C01814=1078.084,-56.704,-56.750,173.466,20.388,153.550
C01815=1078.090,-56.454,-56.762,173.467,20.389,153.550
C01816=1078.097,-56.206,-56.774,173.468,20.391,153.551
C01817=1078.102,-55.955,-56.785,173.470,20.393,153.551
C01818=1078.108,-55.706,-56.797,173.472,20.395,153.551
C01819=1078.115,-55.456,-56.808,173.473,20.397,153.551
C01820=1078.120,-55.206,-56.821,173.475,20.398,153.551
C01821=1078.126,-54.957,-56.832,173.476,20.400,153.551
C01822=1078.133,-54.707,-56.844,173.478,20.402,153.551
C01823=1078.138,-54.458,-56.856,173.479,20.404,153.551
C01824=1078.144,-54.208,-56.867,173.480,20.406,153.551
C01825=1078.151,-53.958,-56.879,173.482,20.407,153.551
C01826=1078.157,-53.709,-56.891,173.483,20.409,153.552
C01827=1078.163,-53.459,-56.902,173.485,20.411,153.552
C01828=1078.169,-53.209,-56.914,173.486,20.413,153.552
C01829=1078.175,-52.960,-56.926,173.488,20.415,153.552
C01830=1078.181,-52.710,-56.938,173.489,20.417,153.552
C01831=1078.188,-52.460,-56.950,173.491,20.419,153.552
C01832=1078.194,-52.211,-56.961,173.492,20.420,153.552
C01833=1078.199,-51.961,-56.973,173.494,20.422,153.552
C01834=1078.206,-51.711,-56.985,173.495,20.424,153.552
C01835=1078.212,-51.462,-56.997,173.496,20.426,153.553
C01836=1078.218,-51.212,-57.009,173.498,20.428,153.553
C01837=1078.224,-50.962,-57.021,173.499,20.429,153.553
C01838=1078.230,-50.712,-57.033,173.500,20.431,153.553
C01839=1078.236,-50.464,-57.045,173.502,20.433,153.553
C01840=1078.243,-50.213,-57.056,173.504,20.435,153.553
C01841=1078.248,-49.964,-57.068,173.505,20.437,153.553
C01842=1078.255,-49.689,-57.082,173.507,20.439,153.553
C01843=1078.262,-49.415,-57.095,173.508,20.441,153.554
C01844=1078.268,-49.141,-57.108,173.510,20.443,153.554
C01845=1078.274,-48.866,-57.121,173.511,20.445,153.554
C01846=1078.281,-48.616,-57.133,173.513,20.447,153.554
C01847=1078.286,-48.367,-57.145,173.514,20.449,153.554
C01848=1078.292,-48.117,-57.157,173.516,20.451,153.554
C01849=1078.298,-47.867,-57.169,173.517,20.453,153.554
C01850=1078.304,-47.618,-57.181,173.518,20.455,153.554
C01851=1078.310,-47.368,-57.194,173.520,20.457,153.555
C01852=1078.316,-47.118,-57.206,173.522,20.459,153.555
C01853=1078.321,-46.869,-57.217,173.523,20.461,153.555
C01854=1078.328,-46.619,-57.229,173.524,20.463,153.555
C01855=1078.334,-46.369,-57.242,173.526,20.465,153.555
C01856=1078.339,-46.120,-57.254,173.527,20.467,153.555
C01857=1078.346,-45.870,-57.266,173.529,20.468,153.555
C01858=1078.352,-45.621,-57.279,173.530,20.470,153.555
C01859=1078.357,-45.371,-57.291,173.531,20.472,153.556
C01860=1078.363,-45.121,-57.302,173.533,20.474,153.556
C01861=1078.369,-44.871,-57.315,173.535,20.476,153.556
C01862=1078.375,-44.622,-57.327,173.536,20.478,153.556
C01863=1078.381,-44.373,-57.339,173.537,20.480,153.556
C01864=1078.387,-44.123,-57.351,173.539,20.482,153.556
C01865=1078.393,-43.873,-57.364,173.540,20.484,153.556
C01866=1078.399,-43.624,-57.375,173.541,20.486,153.557
C01867=1078.405,-43.374,-57.388,173.543,20.487,153.557
C01868=1078.412,-43.124,-57.400,173.545,20.490,153.557
C01869=1078.417,-42.875,-57.412,173.546,20.492,153.557
C01870=1078.423,-42.625,-57.425,173.548,20.494,153.557
C01871=1078.429,-42.376,-57.437,173.549,20.496,153.557
C01872=1078.435,-42.126,-57.449,173.550,20.498,153.557
C01873=1078.441,-41.877,-57.461,173.552,20.499,153.557
C01874=1078.446,-41.626,-57.473,173.553,20.501,153.558
C01875=1078.453,-41.377,-57.485,173.554,20.503,153.558
C01876=1078.459,-41.127,-57.498,173.556,20.506,153.558
C01877=1078.465,-40.877,-57.510,173.558,20.508,153.558
C01878=1078.471,-40.629,-57.523,173.559,20.510,153.558
C01879=1078.477,-40.379,-57.535,173.560,20.512,153.558
C01880=1078.483,-40.129,-57.548,173.562,20.513,153.558
C01881=1078.490,-39.879,-57.560,173.563,20.515,153.559
C01882=1078.495,-39.630,-57.572,173.564,20.517,153.559
C01883=1078.501,-39.380,-57.584,173.566,20.519,153.559
C01884=1078.507,-39.130,-57.597,173.568,20.521,153.559
C01885=1078.513,-38.881,-57.609,173.569,20.523,153.559
C01886=1078.519,-38.631,-57.622,173.570,20.525,153.559
C01887=1078.525,-38.382,-57.634,173.572,20.527,153.559
C01888=1078.530,-38.132,-57.646,173.573,20.529,153.560
C01889=1078.536,-37.882,-57.659,173.575,20.531,153.560
C01890=1078.542,-37.632,-57.671,173.576,20.533,153.560
C01891=1078.548,-37.383,-57.683,173.577,20.535,153.560
C01892=1078.554,-37.133,-57.696,173.579,20.537,153.560
C01893=1078.560,-36.884,-57.709,173.581,20.539,153.560
C01894=1078.566,-36.634,-57.721,173.582,20.541,153.560
C01895=1078.572,-36.384,-57.734,173.583,20.543,153.561
C01896=1078.578,-36.135,-57.746,173.584,20.545,153.561
C01897=1078.583,-35.885,-57.759,173.586,20.547,153.561
C01898=1078.589,-35.635,-57.771,173.587,20.549,153.561
C01899=1078.595,-35.385,-57.784,173.589,20.552,153.561
C01900=1078.601,-35.136,-57.797,173.591,20.554,153.561
C01901=1078.608,-34.887,-57.809,173.592,20.556,153.562
C01902=1078.613,-34.637,-57.821,173.593,20.558,153.562
C01903=1078.619,-34.388,-57.834,173.594,20.560,153.562
C01904=1078.625,-34.138,-57.846,173.596,20.562,153.562
C01905=1078.631,-33.888,-57.859,173.597,20.564,153.562
C01906=1078.638,-33.614,-57.873,173.599,20.566,153.562
C01907=1078.644,-33.340,-57.887,173.601,20.568,153.563
C01908=1078.651,-33.066,-57.901,173.602,20.571,153.563
C01909=1078.657,-32.792,-57.914,173.604,20.573,153.563
C01910=1078.663,-32.542,-57.927,173.605,20.575,153.563
C01911=1078.669,-32.293,-57.940,173.606,20.577,153.563
C01912=1078.675,-32.043,-57.953,173.608,20.579,153.563
C01913=1078.681,-31.793,-57.965,173.609,20.581,153.564
C01914=1078.686,-31.544,-57.978,173.611,20.583,153.564
C01915=1078.693,-31.294,-57.991,173.612,20.585,153.564
C01916=1078.698,-31.045,-58.003,173.614,20.587,153.564
C01917=1078.704,-30.795,-58.016,173.615,20.589,153.564
C01918=1078.711,-30.545,-58.029,173.616,20.591,153.564
C01919=1078.716,-30.296,-58.042,173.618,20.593,153.565
C01920=1078.722,-30.046,-58.054,173.619,20.595,153.565
C01921=1078.729,-29.796,-58.068,173.621,20.598,153.565
C01922=1078.734,-29.546,-58.080,173.622,20.600,153.565
C01923=1078.740,-29.297,-58.092,173.624,20.602,153.565
C01924=1078.747,-29.048,-58.105,173.625,20.604,153.565
C01925=1078.753,-28.798,-58.118,173.626,20.606,153.566
C01926=1078.759,-28.549,-58.130,173.628,20.608,153.566
C01927=1078.765,-28.299,-58.143,173.630,20.610,153.566
C01928=1078.771,-28.049,-58.156,173.631,20.612,153.566
C01929=1078.777,-27.800,-58.168,173.632,20.614,153.566
C01930=1078.783,-27.550,-58.182,173.634,20.616,153.566
C01931=1078.789,-27.300,-58.194,173.635,20.618,153.566
C01932=1078.795,-27.051,-58.208,173.636,20.620,153.567
C01933=1078.800,-26.801,-58.221,173.638,20.622,153.567
C01934=1078.806,-26.551,-58.233,173.640,20.624,153.567
C01935=1078.812,-26.302,-58.247,173.641,20.626,153.567
C01936=1078.818,-26.053,-58.259,173.642,20.629,153.567
C01937=1078.824,-25.803,-58.272,173.643,20.631,153.568
C01938=1078.830,-25.553,-58.285,173.645,20.633,153.568
C01939=1078.835,-25.304,-58.298,173.646,20.635,153.568
C01940=1078.841,-25.054,-58.311,173.648,20.637,153.568
C01941=1078.847,-24.805,-58.324,173.650,20.639,153.568
C01942=1078.853,-24.555,-58.337,173.651,20.641,153.568
C01943=1078.859,-24.306,-58.350,173.652,20.643,153.568
C01944=1078.865,-24.055,-58.363,173.653,20.646,153.569
C01945=1078.871,-23.806,-58.376,173.655,20.648,153.569
C01946=1078.877,-23.556,-58.389,173.657,20.650,153.569
C01947=1078.883,-23.307,-58.402,173.658,20.652,153.569
C01948=1078.889,-23.057,-58.415,173.659,20.654,153.569
C01949=1078.894,-22.808,-58.429,173.661,20.656,153.570
C01950=1078.900,-22.558,-58.441,173.662,20.658,153.570
C01951=1078.906,-22.308,-58.455,173.663,20.661,153.570
C01952=1078.912,-22.059,-58.467,173.665,20.663,153.570
C01953=1078.918,-21.810,-58.480,173.666,20.665,153.570
C01954=1078.923,-21.560,-58.493,173.668,20.667,153.571
C01955=1078.929,-21.310,-58.506,173.669,20.669,153.571
C01956=1078.935,-21.061,-58.519,173.670,20.671,153.571
C01957=1078.941,-20.811,-58.532,173.673,20.673,153.571
C01958=1078.947,-20.562,-58.546,173.674,20.676,153.571
C01959=1078.953,-20.312,-58.559,173.675,20.678,153.571
C01960=1078.959,-20.063,-58.572,173.676,20.680,153.572
C01961=1078.965,-19.813,-58.585,173.678,20.682,153.572
C01962=1078.970,-19.563,-58.598,173.679,20.684,153.572
C01963=1078.977,-19.314,-58.612,173.681,20.686,153.572
C01964=1078.983,-19.064,-58.624,173.682,20.689,153.572
C01965=1078.989,-18.814,-58.638,173.683,20.691,153.573
C01966=1078.995,-18.564,-58.652,173.685,20.693,153.573
C01967=1079.001,-18.315,-58.664,173.686,20.695,153.573
C01968=1079.007,-18.065,-58.678,173.687,20.697,153.573
C01969=1079.013,-17.816,-58.691,173.690,20.699,153.573
C01970=1079.019,-17.541,-58.706,173.691,20.702,153.573
C01971=1079.026,-17.266,-58.721,173.692,20.704,153.574
C01972=1079.033,-16.991,-58.735,173.694,20.706,153.574
C01973=1079.039,-16.716,-58.749,173.695,20.709,153.574
C01974=1079.045,-16.466,-58.762,173.696,20.711,153.574
C01975=1079.051,-16.217,-58.776,173.699,20.713,153.574
C01976=1079.057,-15.968,-58.789,173.700,20.715,153.574
C01977=1079.063,-15.718,-58.802,173.701,20.717,153.575
C01978=1079.069,-15.468,-58.815,173.702,20.719,153.575
C01979=1079.074,-15.219,-58.829,173.704,20.721,153.575
C01980=1079.081,-14.970,-58.842,173.705,20.723,153.575
C01981=1079.086,-14.719,-58.855,173.707,20.726,153.575
C01982=1079.092,-14.470,-58.869,173.708,20.728,153.576
C01983=1079.098,-14.221,-58.882,173.710,20.730,153.576
C01984=1079.104,-13.971,-58.896,173.711,20.732,153.576
C01985=1079.110,-13.722,-58.909,173.712,20.734,153.576
C01986=1079.115,-13.472,-58.922,173.714,20.737,153.576
C01987=1079.122,-13.222,-58.936,173.715,20.739,153.577
C01988=1079.127,-12.972,-58.950,173.717,20.741,153.577
C01989=1079.134,-12.723,-58.963,173.718,20.743,153.577
C01990=1079.139,-12.473,-58.977,173.719,20.746,153.577
C01991=1079.145,-12.224,-58.989,173.721,20.748,153.577
C01992=1079.150,-11.974,-59.003,173.723,20.750,153.578
C01993=1079.157,-11.725,-59.017,173.724,20.752,153.578
C01994=1079.162,-11.475,-59.030,173.725,20.755,153.578
C01995=1079.168,-11.226,-59.044,173.726,20.757,153.578
C01996=1079.174,-10.976,-59.058,173.728,20.759,153.578
C01997=1079.180,-10.727,-59.071,173.730,20.761,153.578
C01998=1079.186,-10.477,-59.085,173.731,20.763,153.579
C01999=1079.192,-10.227,-59.098,173.732,20.765,153.579
C02000=1079.198,-9.977,-59.111,173.734,20.767,153.579
C02001=1079.204,-9.728,-59.125,173.735,20.770,153.579
C02002=1079.209,-9.478,-59.139,173.737,20.772,153.580
C02003=1079.215,-9.229,-59.152,173.738,20.774,153.580
C02004=1079.221,-8.980,-59.166,173.739,20.776,153.580
C02005=1079.227,-8.730,-59.179,173.741,20.779,153.580
C02006=1079.233,-8.480,-59.193,173.742,20.781,153.580
C02007=1079.239,-8.230,-59.207,173.744,20.783,153.580
C02008=1079.245,-7.981,-59.220,173.745,20.785,153.581
C02009=1079.250,-7.732,-59.234,173.746,20.788,153.581
C02010=1079.257,-7.482,-59.248,173.748,20.790,153.581
C02011=1079.262,-7.233,-59.261,173.749,20.792,153.581
C02012=1079.269,-6.983,-59.275,173.751,20.795,153.582
C02013=1079.274,-6.733,-59.289,173.752,20.797,153.582
C02014=1079.281,-6.484,-59.302,173.754,20.799,153.582
C02015=1079.286,-6.234,-59.316,173.755,20.801,153.582
C02016=1079.292,-5.985,-59.329,173.756,20.803,153.582
C02017=1079.298,-5.735,-59.344,173.758,20.805,153.582
C02018=1079.304,-5.485,-59.357,173.760,20.807,153.583
C02019=1079.310,-5.236,-59.371,173.761,20.809,153.583
C02020=1079.315,-4.986,-59.385,173.762,20.812,153.583
C02021=1079.322,-4.737,-59.398,173.763,20.814,153.583
C02022=1079.328,-4.487,-59.412,173.765,20.816,153.583
C02023=1079.333,-4.237,-59.426,173.767,20.818,153.584
C02024=1079.339,-3.988,-59.439,173.768,20.821,153.584
C02025=1079.345,-3.739,-59.454,173.769,20.823,153.584
C02026=1079.352,-3.489,-59.467,173.770,20.825,153.584
C02027=1079.358,-3.240,-59.481,173.772,20.828,153.584
C02028=1079.363,-2.990,-59.495,173.774,20.830,153.585
C02029=1079.368,-2.740,-59.509,173.775,20.832,153.585
C02030=1079.375,-2.491,-59.522,173.776,20.834,153.585
C02031=1079.380,-2.242,-59.536,173.777,20.836,153.585
C02032=1079.386,-1.991,-59.550,173.779,20.839,153.586
C02033=1079.392,-1.742,-59.565,173.781,20.841,153.586
C02034=1079.398,-1.466,-59.580,173.782,20.844,153.586
C02035=1079.405,-1.190,-59.595,173.784,20.846,153.586
C02036=1079.411,-0.913,-59.611,173.785,20.848,153.586
C02037=1079.417,-0.636,-59.626,173.787,20.851,153.587
C02038=1079.423,-0.387,-59.640,173.788,20.853,153.587
C02039=1079.429,-0.137,-59.655,173.790,20.855,153.587
C02040=1079.435,0.113,-59.668,173.791,20.858,153.587
C02041=1079.441,0.362,-59.682,173.793,20.860,153.587
C02042=1079.447,0.611,-59.696,173.794,20.862,153.588
C02043=1079.453,0.861,-59.711,173.795,20.865,153.588
C02044=1079.458,1.111,-59.724,173.797,20.867,153.588
C02045=1079.464,1.361,-59.738,173.798,20.869,153.588
C02046=1079.469,1.610,-59.753,173.800,20.872,153.589
C02047=1079.476,1.859,-59.766,173.801,20.874,153.589
C02048=1079.482,2.109,-59.780,173.802,20.876,153.589
C02049=1079.487,2.359,-59.794,173.804,20.878,153.589
C02050=1079.493,2.608,-59.809,173.806,20.881,153.589
C02051=1079.498,2.857,-59.823,173.807,20.883,153.590
C02052=1079.504,3.108,-59.837,173.808,20.885,153.590
C02053=1079.510,3.356,-59.851,173.809,20.888,153.590
C02054=1079.516,3.606,-59.865,173.811,20.889,153.590
C02055=1079.523,3.856,-59.879,173.813,20.892,153.590
C02056=1079.528,4.105,-59.894,173.814,20.894,153.591
C02057=1079.534,4.355,-59.907,173.815,20.896,153.591
C02058=1079.539,4.604,-59.921,173.816,20.899,153.591
C02059=1079.546,4.854,-59.936,173.819,20.901,153.591
C02060=1079.551,5.103,-59.950,173.820,20.903,153.591
C02061=1079.557,5.353,-59.964,173.821,20.906,153.592
C02062=1079.563,5.603,-59.979,173.822,20.908,153.592
C02063=1079.568,5.852,-59.993,173.824,20.910,153.592
C02064=1079.575,6.101,-60.006,173.826,20.913,153.592
C02065=1079.581,6.351,-60.021,173.827,20.915,153.592
C02066=1079.587,6.601,-60.035,173.828,20.917,153.593
C02067=1079.592,6.850,-60.049,173.829,20.919,153.593
C02068=1079.598,7.100,-60.064,173.832,20.921,153.593
C02069=1079.604,7.349,-60.078,173.833,20.924,153.593
C02070=1079.610,7.598,-60.092,173.834,20.926,153.594
C02071=1079.616,7.849,-60.106,173.835,20.928,153.594
C02072=1079.622,8.098,-60.121,173.836,20.930,153.594
C02073=1079.627,8.347,-60.135,173.839,20.933,153.594
C02074=1079.633,8.597,-60.150,173.840,20.935,153.594
C02075=1079.639,8.846,-60.164,173.841,20.937,153.595
C02076=1079.645,9.096,-60.179,173.842,20.939,153.595
C02077=1079.651,9.346,-60.192,173.844,20.942,153.595
C02078=1079.656,9.595,-60.207,173.846,20.944,153.595
C02079=1079.663,9.845,-60.221,173.847,20.946,153.595
C02080=1079.669,10.094,-60.235,173.848,20.949,153.596
C02081=1079.675,10.344,-60.249,173.850,20.951,153.596
C02082=1079.681,10.593,-60.264,173.851,20.954,153.596
C02083=1079.686,10.842,-60.278,173.853,20.956,153.596
C02084=1079.693,11.092,-60.293,173.854,20.958,153.596
C02085=1079.698,11.342,-60.307,173.855,20.960,153.597
C02086=1079.705,11.591,-60.322,173.857,20.962,153.597
C02087=1079.710,11.840,-60.336,173.859,20.964,153.597
C02088=1079.717,12.090,-60.350,173.860,20.967,153.597
C02089=1079.722,12.339,-60.365,173.861,20.969,153.598
C02090=1079.728,12.589,-60.379,173.863,20.971,153.598
C02091=1079.734,12.839,-60.394,173.864,20.974,153.598
C02092=1079.740,13.088,-60.408,173.866,20.976,153.598
C02093=1079.746,13.338,-60.423,173.867,20.978,153.598
C02094=1079.752,13.587,-60.437,173.869,20.981,153.599
C02095=1079.758,13.837,-60.451,173.870,20.983,153.599
C02096=1079.764,14.086,-60.466,173.872,20.985,153.599
C02097=1079.770,14.336,-60.481,173.873,20.987,153.599
C02098=1079.776,14.614,-60.497,173.875,20.989,153.599
C02099=1079.782,14.893,-60.513,173.876,20.992,153.600
C02100=1079.789,15.172,-60.530,173.878,20.995,153.600
C02101=1079.795,15.450,-60.546,173.879,20.997,153.600
C02102=1079.801,15.700,-60.561,173.881,21.000,153.600
C02103=1079.807,15.949,-60.576,173.882,21.002,153.601
C02104=1079.813,16.198,-60.589,173.884,21.004,153.601
C02105=1079.819,16.448,-60.604,173.885,21.006,153.601
C02106=1079.824,16.697,-60.620,173.887,21.009,153.601
C02107=1079.830,16.947,-60.634,173.888,21.011,153.601
C02108=1079.836,17.196,-60.648,173.890,21.014,153.602
C02109=1079.842,17.446,-60.663,173.891,21.016,153.602
C02110=1079.848,17.695,-60.678,173.893,21.018,153.602
C02111=1079.854,17.946,-60.693,173.894,21.021,153.602
C02112=1079.859,18.195,-60.707,173.896,21.022,153.602
C02113=1079.866,18.444,-60.722,173.897,21.025,153.603
C02114=1079.871,18.693,-60.737,173.899,21.027,153.603
C02115=1079.878,18.943,-60.752,173.900,21.030,153.603
C02116=1079.883,19.193,-60.766,173.901,21.032,153.603
C02117=1079.889,19.442,-60.781,173.903,21.034,153.604
C02118=1079.895,19.691,-60.796,173.905,21.037,153.604
C02119=1079.901,19.941,-60.811,173.906,21.039,153.604
C02120=1079.906,20.190,-60.826,173.907,21.041,153.604
C02121=1079.912,20.441,-60.840,173.908,21.043,153.604
C02122=1079.918,20.690,-60.855,173.910,21.046,153.605
C02123=1079.924,20.939,-60.870,173.912,21.048,153.605
C02124=1079.929,21.188,-60.885,173.913,21.050,153.605
C02125=1079.936,21.438,-60.900,173.914,21.053,153.605
C02126=1079.942,21.687,-60.914,173.916,21.055,153.605
C02127=1079.947,21.937,-60.930,173.917,21.057,153.606
C02128=1079.953,22.187,-60.944,173.919,21.059,153.606
C02129=1079.958,22.437,-60.959,173.920,21.062,153.606
C02130=1079.964,22.686,-60.974,173.922,21.064,153.606
C02131=1079.971,22.935,-60.989,173.923,21.067,153.607
C02132=1079.976,23.184,-61.004,173.924,21.069,153.607
C02133=1079.982,23.434,-61.019,173.926,21.071,153.607
C02134=1079.988,23.683,-61.033,173.928,21.074,153.607
C02135=1079.993,23.933,-61.049,173.929,21.076,153.607
C02136=1079.999,24.182,-61.064,173.930,21.078,153.608
C02137=1080.006,24.432,-61.079,173.932,21.080,153.608
C02138=1080.011,24.681,-61.094,173.934,21.083,153.608
C02139=1080.017,24.931,-61.109,173.935,21.085,153.608
C02140=1080.023,25.181,-61.124,173.936,21.087,153.609
C02141=1080.028,25.429,-61.139,173.937,21.089,153.609
C02142=1080.035,25.679,-61.154,173.939,21.092,153.609
C02143=1080.040,25.928,-61.169,173.941,21.094,153.609
C02144=1080.046,26.178,-61.184,173.942,21.096,153.609
C02145=1080.052,26.427,-61.198,173.944,21.099,153.610
C02146=1080.058,26.677,-61.214,173.945,21.101,153.610
C02147=1080.064,26.927,-61.229,173.947,21.103,153.610
C02148=1080.069,27.176,-61.244,173.948,21.106,153.610
C02149=1080.075,27.426,-61.259,173.950,21.108,153.610
C02150=1080.081,27.675,-61.274,173.951,21.110,153.611
C02151=1080.087,27.924,-61.289,173.952,21.112,153.611
C02152=1080.093,28.174,-61.305,173.953,21.115,153.611
C02153=1080.098,28.423,-61.319,173.956,21.117,153.611
C02154=1080.105,28.673,-61.334,173.957,21.119,153.612
C02155=1080.110,28.923,-61.350,173.958,21.122,153.612
C02156=1080.116,29.171,-61.365,173.960,21.124,153.612
C02157=1080.122,29.421,-61.381,173.961,21.127,153.612
C02158=1080.127,29.671,-61.396,173.963,21.129,153.612
C02159=1080.134,29.920,-61.411,173.964,21.131,153.613
C02160=1080.139,30.170,-61.426,173.966,21.134,153.613
C02161=1080.145,30.419,-61.441,173.967,21.136,153.613
C02162=1080.152,30.699,-61.459,173.969,21.138,153.613
C02163=1080.158,30.979,-61.475,173.971,21.141,153.614
C02164=1080.164,31.259,-61.493,173.973,21.144,153.614
C02165=1080.171,31.539,-61.510,173.974,21.146,153.614
C02166=1080.176,31.788,-61.525,173.975,21.148,153.614
C02167=1080.182,32.038,-61.541,173.977,21.151,153.615
C02168=1080.188,32.288,-61.556,173.978,21.153,153.615
C02169=1080.194,32.537,-61.571,173.979,21.156,153.615
C02170=1080.200,32.786,-61.586,173.982,21.158,153.615
C02171=1080.206,33.036,-61.602,173.983,21.160,153.615
C02172=1080.211,33.285,-61.617,173.984,21.162,153.616
C02173=1080.217,33.535,-61.632,173.985,21.164,153.616
C02174=1080.223,33.784,-61.648,173.987,21.167,153.616
C02175=1080.228,34.033,-61.663,173.989,21.169,153.616
C02176=1080.235,34.283,-61.678,173.990,21.172,153.617
C02177=1080.240,34.533,-61.694,173.992,21.174,153.617
C02178=1080.246,34.781,-61.709,173.993,21.177,153.617
C02179=1080.252,35.031,-61.725,173.995,21.179,153.617
C02180=1080.258,35.281,-61.740,173.996,21.181,153.617
C02181=1080.264,35.530,-61.756,173.998,21.184,153.618
C02182=1080.269,35.780,-61.771,173.999,21.185,153.618
C02183=1080.275,36.030,-61.787,174.000,21.188,153.618
C02184=1080.282,36.279,-61.802,174.003,21.190,153.618
C02185=1080.287,36.528,-61.818,174.004,21.192,153.618
C02186=1080.292,36.778,-61.833,174.005,21.195,153.619
C02187=1080.299,37.027,-61.849,174.006,21.197,153.619
C02188=1080.304,37.276,-61.864,174.008,21.200,153.619
C02189=1080.310,37.526,-61.879,174.010,21.202,153.619
C02190=1080.317,37.775,-61.895,174.011,21.204,153.619
C02191=1080.322,38.025,-61.911,174.013,21.207,153.620
C02192=1080.327,38.274,-61.926,174.014,21.208,153.620
C02193=1080.333,38.524,-61.942,174.015,21.211,153.620
C02194=1080.340,38.773,-61.957,174.018,21.213,153.620
C02195=1080.345,39.022,-61.973,174.019,21.216,153.621
C02196=1080.351,39.272,-61.988,174.020,21.218,153.621
C02197=1080.356,39.521,-62.005,174.021,21.220,153.621
C02198=1080.362,39.771,-62.020,174.023,21.223,153.621
C02199=1080.368,40.020,-62.035,174.025,21.225,153.622
C02200=1080.374,40.270,-62.051,174.026,21.227,153.622
C02201=1080.379,40.520,-62.067,174.028,21.230,153.622
C02202=1080.385,40.769,-62.083,174.029,21.232,153.622
C02203=1080.390,41.018,-62.098,174.031,21.234,153.622
C02204=1080.396,41.268,-62.114,174.033,21.237,153.623
C02205=1080.403,41.517,-62.129,174.034,21.239,153.623
C02206=1080.409,41.767,-62.146,174.035,21.241,153.623
C02207=1080.414,42.016,-62.161,174.036,21.243,153.623
C02208=1080.420,42.265,-62.177,174.038,21.246,153.624
C02209=1080.425,42.515,-62.192,174.040,21.248,153.624
C02210=1080.431,42.765,-62.209,174.041,21.251,153.624
C02211=1080.436,43.014,-62.224,174.043,21.253,153.624
C02212=1080.443,43.263,-62.240,174.044,21.255,153.624
C02213=1080.449,43.512,-62.256,174.045,21.257,153.625
C02214=1080.455,43.762,-62.271,174.048,21.260,153.625
C02215=1080.461,44.012,-62.288,174.049,21.262,153.625
C02216=1080.466,44.261,-62.303,174.050,21.264,153.625
C02217=1080.472,44.510,-62.319,174.052,21.267,153.625
C02218=1080.478,44.759,-62.335,174.054,21.269,153.626
C02219=1080.483,45.009,-62.351,174.055,21.272,153.626
C02220=1080.489,45.258,-62.367,174.057,21.274,153.626
C02221=1080.494,45.508,-62.382,174.058,21.276,153.626
C02222=1080.500,45.757,-62.399,174.059,21.278,153.627
C02223=1080.505,46.007,-62.415,174.060,21.281,153.627
C02224=1080.510,46.256,-62.431,174.063,21.283,153.627
C02225=1080.516,46.506,-62.447,174.064,21.286,153.627
C02226=1080.523,46.786,-62.465,174.066,21.289,153.628
C02227=1080.529,47.065,-62.482,174.067,21.291,153.628
C02228=1080.535,47.346,-62.500,174.069,21.294,153.628
C02229=1080.542,47.626,-62.518,174.071,21.297,153.628
C02230=1080.548,47.875,-62.534,174.072,21.298,153.628
C02231=1080.554,48.124,-62.550,174.074,21.301,153.629
C02232=1080.560,48.373,-62.567,174.075,21.303,153.629
C02233=1080.565,48.623,-62.582,174.077,21.306,153.629
C02234=1080.570,48.873,-62.599,174.078,21.308,153.629
C02235=1080.576,49.122,-62.615,174.079,21.310,153.630
C02236=1080.582,49.372,-62.631,174.082,21.313,153.630
C02237=1080.587,49.621,-62.647,174.083,21.315,153.630
C02238=1080.593,49.870,-62.663,174.084,21.317,153.630
C02239=1080.599,50.120,-62.679,174.086,21.319,153.630
C02240=1080.605,50.369,-62.695,174.087,21.322,153.631
C02241=1080.611,50.619,-62.711,174.089,21.324,153.631
C02242=1080.617,50.868,-62.727,174.091,21.327,153.631
C02243=1080.622,51.118,-62.744,174.092,21.329,153.631
C02244=1080.627,51.367,-62.760,174.093,21.331,153.632
C02245=1080.633,51.616,-62.776,174.096,21.334,153.632
C02246=1080.639,51.866,-62.792,174.097,21.336,153.632
C02247=1080.645,52.115,-62.808,174.098,21.338,153.632
C02248=1080.651,52.365,-62.824,174.100,21.340,153.632
C02249=1080.657,52.614,-62.840,174.101,21.343,153.633
C02250=1080.663,52.863,-62.857,174.103,21.345,153.633
C02251=1080.668,53.113,-62.874,174.105,21.348,153.633
C02252=1080.674,53.362,-62.890,174.106,21.350,153.633
C02253=1080.679,53.612,-62.905,174.107,21.352,153.633
C02254=1080.685,53.861,-62.921,174.109,21.355,153.634
C02255=1080.691,54.110,-62.938,174.111,21.356,153.634
C02256=1080.697,54.360,-62.954,174.112,21.359,153.634
C02257=1080.702,54.609,-62.971,174.114,21.361,153.634
C02258=1080.708,54.859,-62.987,174.115,21.363,153.634
C02259=1080.714,55.108,-63.003,174.117,21.366,153.635
C02260=1080.720,55.357,-63.019,174.119,21.368,153.635
C02261=1080.726,55.607,-63.036,174.120,21.370,153.635
C02262=1080.732,55.856,-63.052,174.121,21.373,153.635
C02263=1080.737,56.106,-63.069,174.123,21.375,153.636
C02264=1080.743,56.355,-63.085,174.125,21.377,153.636
C02265=1080.749,56.604,-63.101,174.127,21.380,153.636
C02266=1080.755,56.854,-63.118,174.128,21.382,153.636
C02267=1080.761,57.103,-63.134,174.129,21.384,153.636
C02268=1080.766,57.353,-63.151,174.132,21.387,153.637
C02269=1080.772,57.602,-63.167,174.133,21.389,153.637
C02270=1080.778,57.851,-63.183,174.134,21.391,153.637
C02271=1080.784,58.101,-63.199,174.136,21.393,153.637
C02272=1080.790,58.350,-63.216,174.138,21.395,153.637
C02273=1080.795,58.600,-63.233,174.139,21.398,153.638
C02274=1080.801,58.849,-63.249,174.141,21.400,153.638
C02275=1080.807,59.098,-63.265,174.142,21.402,153.638
C02276=1080.813,59.348,-63.281,174.143,21.405,153.638
C02277=1080.819,59.597,-63.298,174.146,21.407,153.638
C02278=1080.824,59.847,-63.314,174.147,21.409,153.639
C02279=1080.830,60.096,-63.331,174.148,21.411,153.639
C02280=1080.836,60.345,-63.348,174.150,21.414,153.639
C02281=1080.842,60.594,-63.364,174.152,21.416,153.639
C02282=1080.847,60.844,-63.381,174.153,21.418,153.639
C02283=1080.853,61.093,-63.397,174.155,21.421,153.640
C02284=1080.859,61.343,-63.413,174.156,21.423,153.640
C02285=1080.865,61.592,-63.430,174.159,21.425,153.640
C02286=1080.870,61.842,-63.446,174.160,21.427,153.640
C02287=1080.877,62.090,-63.463,174.161,21.429,153.640
C02288=1080.883,62.340,-63.480,174.163,21.432,153.641
C02289=1080.889,62.590,-63.496,174.165,21.434,153.641
C02290=1080.896,62.870,-63.515,174.167,21.437,153.641
C02291=1080.901,63.149,-63.534,174.168,21.439,153.641
C02292=1080.908,63.429,-63.552,174.170,21.441,153.641
C02293=1080.915,63.709,-63.571,174.172,21.444,153.642
C02294=1080.920,63.958,-63.587,174.173,21.446,153.642
C02295=1080.927,64.207,-63.604,174.175,21.448,153.642
C02296=1080.933,64.457,-63.621,174.177,21.451,153.642
C02297=1080.939,64.707,-63.638,174.178,21.453,153.642
C02298=1080.944,64.956,-63.654,174.179,21.455,153.643
C02299=1080.950,65.205,-63.671,174.182,21.457,153.643
C02300=1080.956,65.454,-63.688,174.183,21.459,153.643
C02301=1080.961,65.704,-63.704,174.184,21.462,153.643
C02302=1080.967,65.953,-63.721,174.186,21.464,153.643
C02303=1080.973,66.202,-63.738,174.188,21.466,153.644
C02304=1080.979,66.452,-63.755,174.190,21.469,153.644
C02305=1080.984,66.701,-63.771,174.191,21.471,153.644
C02306=1080.990,66.950,-63.788,174.192,21.473,153.644
C02307=1080.995,67.200,-63.805,174.194,21.476,153.644
C02308=1081.002,67.450,-63.822,174.196,21.478,153.645
C02309=1081.007,67.699,-63.839,174.197,21.480,153.645
C02310=1081.013,67.948,-63.856,174.199,21.483,153.645
C02311=1081.019,68.197,-63.873,174.201,21.485,153.645
C02312=1081.025,68.447,-63.889,174.203,21.487,153.645
C02313=1081.030,68.696,-63.906,174.204,21.489,153.646
C02314=1081.036,68.945,-63.923,174.205,21.491,153.646
C02315=1081.041,69.195,-63.940,174.207,21.494,153.646
C02316=1081.048,69.443,-63.957,174.209,21.496,153.646
C02317=1081.053,69.694,-63.974,174.211,21.499,153.646
C02318=1081.059,69.943,-63.991,174.212,21.500,153.647
C02319=1081.065,70.192,-64.008,174.214,21.502,153.647
C02320=1081.070,70.442,-64.025,174.216,21.505,153.647
C02321=1081.076,70.690,-64.042,174.217,21.507,153.647
C02322=1081.082,70.940,-64.059,174.218,21.509,153.647
C02323=1081.087,71.189,-64.076,174.220,21.512,153.648
C02324=1081.094,71.439,-64.093,174.222,21.514,153.648
C02325=1081.099,71.688,-64.111,174.224,21.516,153.648
C02326=1081.104,71.938,-64.127,174.225,21.518,153.648
C02327=1081.111,72.187,-64.144,174.226,21.521,153.648
C02328=1081.116,72.436,-64.161,174.229,21.523,153.649
C02329=1081.121,72.685,-64.179,174.230,21.525,153.649
C02330=1081.127,72.935,-64.195,174.232,21.528,153.649
C02331=1081.133,73.184,-64.213,174.233,21.530,153.649
C02332=1081.139,73.434,-64.230,174.235,21.532,153.649
C02333=1081.145,73.683,-64.247,174.237,21.535,153.650
C02334=1081.150,73.933,-64.264,174.238,21.537,153.650
C02335=1081.156,74.182,-64.281,174.240,21.539,153.650
C02336=1081.162,74.432,-64.299,174.242,21.541,153.650
C02337=1081.168,74.681,-64.315,174.243,21.544,153.650
C02338=1081.173,74.930,-64.333,174.245,21.546,153.650
C02339=1081.179,75.179,-64.350,174.246,21.548,153.651
C02340=1081.185,75.428,-64.367,174.249,21.550,153.651
C02341=1081.191,75.678,-64.384,174.250,21.553,153.651
C02342=1081.196,75.927,-64.402,174.251,21.555,153.651
C02343=1081.202,76.177,-64.419,174.253,21.557,153.651
C02344=1081.208,76.426,-64.435,174.255,21.559,153.652
C02345=1081.213,76.675,-64.453,174.257,21.562,153.652
C02346=1081.219,76.925,-64.471,174.258,21.564,153.652
C02347=1081.224,77.174,-64.488,174.259,21.566,153.652
C02348=1081.231,77.423,-64.505,174.262,21.568,153.652
C02349=1081.236,77.672,-64.522,174.263,21.570,153.652
C02350=1081.242,77.922,-64.540,174.265,21.573,153.653
C02351=1081.248,78.171,-64.557,174.266,21.575,153.653
C02352=1081.253,78.421,-64.575,174.268,21.577,153.653
C02353=1081.259,78.669,-64.592,174.270,21.579,153.653
C02354=1081.265,78.949,-64.611,174.272,21.582,153.653
C02355=1081.271,79.229,-64.630,174.273,21.584,153.654
C02356=1081.278,79.508,-64.650,174.275,21.587,153.654
C02357=1081.284,79.788,-64.669,174.277,21.590,153.654
C02358=1081.290,80.038,-64.687,174.279,21.592,153.654
C02359=1081.296,80.287,-64.705,174.281,21.594,153.655
C02360=1081.302,80.536,-64.722,174.282,21.596,153.655
C02361=1081.307,80.786,-64.739,174.284,21.598,153.655
C02362=1081.313,81.036,-64.757,174.286,21.601,153.655
C02363=1081.318,81.285,-64.775,174.287,21.603,153.655
C02364=1081.324,81.534,-64.792,174.289,21.605,153.655
C02365=1081.329,81.783,-64.810,174.290,21.608,153.656
C02366=1081.335,82.033,-64.827,174.292,21.609,153.656
C02367=1081.341,82.282,-64.845,174.294,21.612,153.656
C02368=1081.346,82.531,-64.862,174.295,21.614,153.656
C02369=1081.352,82.781,-64.880,174.298,21.616,153.656
C02370=1081.358,83.030,-64.898,174.299,21.619,153.657
C02371=1081.363,83.279,-64.915,174.301,21.621,153.657
C02372=1081.369,83.528,-64.933,174.302,21.623,153.657
C02373=1081.376,83.777,-64.950,174.304,21.625,153.657
C02374=1081.381,84.027,-64.967,174.306,21.628,153.657
C02375=1081.387,84.276,-64.985,174.307,21.630,153.658
C02376=1081.393,84.526,-65.003,174.309,21.632,153.658
C02377=1081.398,84.775,-65.020,174.311,21.634,153.658
C02378=1081.404,85.024,-65.038,174.313,21.636,153.658
C02379=1081.410,85.274,-65.056,174.314,21.638,153.658
C02380=1081.415,85.523,-65.073,174.315,21.641,153.659
C02381=1081.421,85.772,-65.091,174.318,21.643,153.659
C02382=1081.427,86.022,-65.109,174.319,21.645,153.659
C02383=1081.432,86.271,-65.126,174.321,21.647,153.659
C02384=1081.438,86.520,-65.144,174.323,21.649,153.659
C02385=1081.443,86.770,-65.162,174.325,21.652,153.659
C02386=1081.449,87.019,-65.180,174.326,21.654,153.660
C02387=1081.455,87.268,-65.198,174.328,21.657,153.660
C02388=1081.461,87.517,-65.215,174.330,21.658,153.660
C02389=1081.466,87.767,-65.233,174.331,21.660,153.660
C02390=1081.472,88.016,-65.251,174.333,21.663,153.660
C02391=1081.478,88.265,-65.268,174.335,21.665,153.660
C02392=1081.484,88.515,-65.286,174.337,21.667,153.660
C02393=1081.489,88.764,-65.304,174.338,21.669,153.661
C02394=1081.495,89.013,-65.322,174.340,21.672,153.661
C02395=1081.501,89.263,-65.339,174.342,21.674,153.661
C02396=1081.506,89.512,-65.357,174.344,21.676,153.661
C02397=1081.513,89.761,-65.376,174.345,21.678,153.661
C02398=1081.518,90.010,-65.393,174.347,21.680,153.662
C02399=1081.525,90.260,-65.411,174.349,21.682,153.662
C02400=1081.530,90.509,-65.429,174.350,21.684,153.662
C02401=1081.536,90.758,-65.446,174.352,21.687,153.662
C02402=1081.542,91.008,-65.464,174.354,21.689,153.662
C02403=1081.546,91.257,-65.482,174.356,21.691,153.662
C02404=1081.553,91.507,-65.500,174.357,21.693,153.663
C02405=1081.558,91.755,-65.519,174.359,21.696,153.663
C02406=1081.564,92.004,-65.536,174.361,21.698,153.663
C02407=1081.569,92.254,-65.555,174.363,21.700,153.663
C02408=1081.575,92.503,-65.572,174.364,21.702,153.663
C02409=1081.581,92.753,-65.590,174.366,21.704,153.663
C02410=1081.587,93.001,-65.608,174.368,21.707,153.664
C02411=1081.592,93.251,-65.627,174.369,21.709,153.664
C02412=1081.598,93.501,-65.645,174.371,21.711,153.664
C02413=1081.603,93.750,-65.662,174.373,21.713,153.664
C02414=1081.609,94.000,-65.681,174.375,21.715,153.664
C02415=1081.614,94.248,-65.699,174.376,21.717,153.664
C02416=1081.621,94.498,-65.717,174.379,21.720,153.665
C02417=1081.626,94.747,-65.734,174.380,21.722,153.665
C02418=1081.632,95.026,-65.755,174.382,21.725,153.665
C02419=1081.639,95.307,-65.776,174.384,21.727,153.665
C02420=1081.644,95.586,-65.796,174.386,21.729,153.665
C02421=1081.652,95.866,-65.816,174.388,21.732,153.666
C02422=1081.657,96.115,-65.835,174.390,21.734,153.666
C02423=1081.662,96.364,-65.853,174.391,21.736,153.666
C02424=1081.668,96.614,-65.871,174.393,21.738,153.666
C02425=1081.674,96.862,-65.889,174.395,21.740,153.666
C02426=1081.680,97.112,-65.907,174.397,21.743,153.666
C02427=1081.685,97.361,-65.925,174.398,21.745,153.667
C02428=1081.692,97.610,-65.944,174.401,21.747,153.667
C02429=1081.697,97.860,-65.962,174.402,21.749,153.667
C02430=1081.703,98.109,-65.980,174.404,21.751,153.667
C02431=1081.709,98.358,-65.998,174.406,21.753,153.667
C02432=1081.714,98.608,-66.016,174.408,21.755,153.667
C02433=1081.720,98.857,-66.035,174.409,21.757,153.667
C02434=1081.725,99.106,-66.053,174.411,21.760,153.668
C02435=1081.731,99.355,-66.072,174.413,21.762,153.668
C02436=1081.737,99.604,-66.089,174.414,21.764,153.668
C02437=1081.742,99.854,-66.108,174.416,21.766,153.668
C02438=1081.748,100.103,-66.126,174.418,21.768,153.668
C02439=1081.754,100.353,-66.144,174.420,21.770,153.668
C02440=1081.760,100.602,-66.163,174.421,21.772,153.669
C02441=1081.765,100.851,-66.181,174.424,21.775,153.669
C02442=1081.772,101.100,-66.200,174.425,21.776,153.669
C02443=1081.777,101.350,-66.218,174.427,21.779,153.669
C02444=1081.783,101.599,-66.236,174.429,21.781,153.669
C02445=1081.788,101.848,-66.255,174.431,21.784,153.669
C02446=1081.794,102.098,-66.274,174.432,21.786,153.670
C02447=1081.799,102.347,-66.291,174.434,21.788,153.670
C02448=1081.805,102.596,-66.311,174.436,21.790,153.670
C02449=1081.811,102.844,-66.329,174.438,21.792,153.670
C02450=1081.816,103.094,-66.347,174.439,21.794,153.670
C02451=1081.822,103.344,-66.366,174.442,21.796,153.670
C02452=1081.827,103.593,-66.384,174.443,21.798,153.671
C02453=1081.834,103.842,-66.403,174.445,21.801,153.671
C02454=1081.838,104.091,-66.421,174.446,21.803,153.671
C02455=1081.844,104.341,-66.440,174.449,21.805,153.671
C02456=1081.850,104.589,-66.459,174.450,21.807,153.671
C02457=1081.855,104.839,-66.477,174.452,21.809,153.671
C02458=1081.862,105.088,-66.496,174.454,21.811,153.672
C02459=1081.867,105.337,-66.515,174.456,21.814,153.672
C02460=1081.873,105.587,-66.533,174.458,21.816,153.672
C02461=1081.878,105.836,-66.552,174.460,21.818,153.672
C02462=1081.884,106.085,-66.571,174.462,21.820,153.672
C02463=1081.890,106.335,-66.589,174.463,21.822,153.672
C02464=1081.895,106.584,-66.608,174.465,21.824,153.672
C02465=1081.901,106.833,-66.626,174.467,21.826,153.673
C02466=1081.907,107.083,-66.645,174.469,21.829,153.673
C02467=1081.912,107.331,-66.664,174.470,21.831,153.673
C02468=1081.918,107.581,-66.682,174.473,21.833,153.673
C02469=1081.924,107.830,-66.702,174.474,21.835,153.673
C02470=1081.929,108.079,-66.720,174.476,21.837,153.673
C02471=1081.935,108.328,-66.738,174.478,21.839,153.674
C02472=1081.941,108.578,-66.758,174.480,21.842,153.674
C02473=1081.947,108.826,-66.776,174.481,21.843,153.674
C02474=1081.952,109.076,-66.794,174.484,21.845,153.674
C02475=1081.958,109.326,-66.814,174.485,21.847,153.674
C02476=1081.963,109.574,-66.832,174.487,21.850,153.674
C02477=1081.969,109.824,-66.851,174.489,21.852,153.674
C02478=1081.975,110.073,-66.870,174.491,21.854,153.674
C02479=1081.980,110.322,-66.888,174.492,21.856,153.675
C02480=1081.986,110.572,-66.907,174.495,21.858,153.675
C02481=1081.992,110.821,-66.926,174.496,21.860,153.675
C02482=1081.998,111.100,-66.948,174.498,21.862,153.675
C02483=1082.005,111.380,-66.968,174.500,21.865,153.675
C02484=1082.011,111.660,-66.990,174.503,21.867,153.675
C02485=1082.018,111.940,-67.010,174.505,21.869,153.676
C02486=1082.023,112.189,-67.029,174.506,21.871,153.676
C02487=1082.029,112.438,-67.049,174.509,21.874,153.676
C02488=1082.034,112.688,-67.068,174.511,21.876,153.676
C02489=1082.039,112.936,-67.087,174.512,21.878,153.676
C02490=1082.046,113.186,-67.105,174.514,21.880,153.676
C02491=1082.052,113.435,-67.125,174.516,21.882,153.676
C02492=1082.057,113.684,-67.144,174.518,21.884,153.676
C02493=1082.062,113.933,-67.163,174.520,21.886,153.677
C02494=1082.068,114.183,-67.182,174.522,21.888,153.677
C02495=1082.074,114.432,-67.201,174.523,21.890,153.677
C02496=1082.080,114.681,-67.220,174.525,21.893,153.677
C02497=1082.085,114.930,-67.239,174.527,21.895,153.677
C02498=1082.091,115.179,-67.258,174.529,21.897,153.677
C02499=1082.097,115.429,-67.277,174.531,21.899,153.678
C02500=1082.102,115.677,-67.296,174.533,21.901,153.678
C02501=1082.107,115.927,-67.315,174.535,21.904,153.678
C02502=1082.113,116.176,-67.335,174.536,21.905,153.678
C02503=1082.118,116.425,-67.353,174.539,21.908,153.678
C02504=1082.124,116.674,-67.373,174.540,21.910,153.678
C02505=1082.130,116.924,-67.392,174.542,21.912,153.678
C02506=1082.135,117.173,-67.411,174.544,21.914,153.679
C02507=1082.140,117.422,-67.430,174.546,21.916,153.679
C02508=1082.146,117.671,-67.449,174.548,21.918,153.679
C02509=1082.152,117.921,-67.469,174.550,21.920,153.679
C02510=1082.157,118.170,-67.488,174.552,21.922,153.679
C02511=1082.162,118.419,-67.507,174.553,21.924,153.679
C02512=1082.168,118.668,-67.527,174.556,21.927,153.679
C02513=1082.174,118.917,-67.546,174.557,21.929,153.680
C02514=1082.180,119.167,-67.565,174.559,21.931,153.680
C02515=1082.185,119.415,-67.584,174.561,21.933,153.680
C02516=1082.191,119.665,-67.603,174.563,21.935,153.680
C02517=1082.196,119.914,-67.623,174.565,21.937,153.680
C02518=1082.202,120.164,-67.642,174.567,21.939,153.680
C02519=1082.208,120.413,-67.662,174.569,21.941,153.680
C02520=1082.213,120.661,-67.681,174.570,21.943,153.681
C02521=1082.218,120.911,-67.700,174.573,21.946,153.681
C02522=1082.224,121.161,-67.720,174.575,21.948,153.681
C02523=1082.230,121.409,-67.740,174.576,21.949,153.681
C02524=1082.235,121.659,-67.759,174.579,21.952,153.681
C02525=1082.241,121.908,-67.778,174.580,21.954,153.681
C02526=1082.246,122.157,-67.797,174.582,21.956,153.681
C02527=1082.252,122.406,-67.817,174.584,21.958,153.681
C02528=1082.258,122.655,-67.836,174.586,21.960,153.682
C02529=1082.264,122.905,-67.855,174.588,21.962,153.682
C02530=1082.269,123.154,-67.875,174.590,21.964,153.682
C02531=1082.275,123.403,-67.895,174.592,21.966,153.682
C02532=1082.281,123.652,-67.914,174.594,21.969,153.682
C02533=1082.286,123.901,-67.933,174.596,21.970,153.682
C02534=1082.292,124.150,-67.953,174.598,21.972,153.682
C02535=1082.297,124.400,-67.973,174.599,21.974,153.682
C02536=1082.303,124.649,-67.992,174.602,21.977,153.683
C02537=1082.309,124.898,-68.012,174.604,21.979,153.683
C02538=1082.314,125.147,-68.031,174.605,21.980,153.683
C02539=1082.320,125.397,-68.050,174.608,21.983,153.683
C02540=1082.326,125.645,-68.070,174.609,21.985,153.683
C02541=1082.332,125.895,-68.089,174.611,21.987,153.683
C02542=1082.338,126.144,-68.109,174.614,21.989,153.683
C02543=1082.342,126.393,-68.129,174.615,21.991,153.683
C02544=1082.348,126.642,-68.148,174.617,21.993,153.684
C02545=1082.354,126.891,-68.168,174.619,21.994,153.684
C02546=1082.361,127.171,-68.190,174.621,21.997,153.684
C02547=1082.367,127.451,-68.212,174.624,21.999,153.684
C02548=1082.373,127.731,-68.234,174.626,22.001,153.684
C02549=1082.379,128.010,-68.256,174.628,22.004,153.684
C02550=1082.385,128.259,-68.276,174.630,22.006,153.684
C02551=1082.391,128.508,-68.296,174.632,22.008,153.684
C02552=1082.397,128.758,-68.315,174.634,22.010,153.684
C02553=1082.403,129.006,-68.335,174.636,22.012,153.685
C02554=1082.408,129.256,-68.354,174.638,22.014,153.685
C02555=1082.413,129.505,-68.375,174.640,22.016,153.685
C02556=1082.419,129.754,-68.394,174.642,22.018,153.685
C02557=1082.425,130.003,-68.414,174.644,22.020,153.685
C02558=1082.431,130.253,-68.433,174.646,22.022,153.685
C02559=1082.437,130.501,-68.453,174.648,22.024,153.685
C02560=1082.442,130.751,-68.474,174.650,22.026,153.685
C02561=1082.448,131.000,-68.493,174.652,22.028,153.685
C02562=1082.454,131.249,-68.513,174.654,22.029,153.685
C02563=1082.459,131.498,-68.532,174.656,22.032,153.686
C02564=1082.465,131.747,-68.552,174.658,22.034,153.686
C02565=1082.471,131.997,-68.573,174.660,22.036,153.686
C02566=1082.477,132.246,-68.592,174.662,22.038,153.686
C02567=1082.483,132.495,-68.612,174.664,22.040,153.686
C02568=1082.488,132.745,-68.632,174.666,22.042,153.686
C02569=1082.494,132.994,-68.652,174.668,22.044,153.686
C02570=1082.499,133.242,-68.672,174.670,22.046,153.686
C02571=1082.504,133.491,-68.691,174.672,22.048,153.686
C02572=1082.510,133.740,-68.711,174.675,22.050,153.687
C02573=1082.516,133.990,-68.732,174.676,22.052,153.687
C02574=1082.522,134.239,-68.752,174.678,22.054,153.687
C02575=1082.527,134.489,-68.772,174.681,22.056,153.687
C02576=1082.533,134.738,-68.792,174.682,22.058,153.687
C02577=1082.539,134.986,-68.812,174.684,22.060,153.687
C02578=1082.544,135.235,-68.833,174.686,22.062,153.687
C02579=1082.550,135.485,-68.852,174.688,22.064,153.687
C02580=1082.555,135.734,-68.872,174.690,22.066,153.688
C02581=1082.561,135.983,-68.892,174.692,22.068,153.688
C02582=1082.567,136.232,-68.913,174.694,22.070,153.688
C02583=1082.572,136.481,-68.932,174.697,22.072,153.688
C02584=1082.578,136.730,-68.952,174.698,22.074,153.688
C02585=1082.583,136.979,-68.973,174.700,22.076,153.688
C02586=1082.589,137.228,-68.993,174.703,22.078,153.688
C02587=1082.595,137.477,-69.013,174.704,22.080,153.688
C02588=1082.600,137.727,-69.032,174.706,22.082,153.688
C02589=1082.606,137.976,-69.053,174.709,22.084,153.688
C02590=1082.612,138.225,-69.073,174.710,22.086,153.689
C02591=1082.617,138.474,-69.094,174.713,22.088,153.689
C02592=1082.623,138.723,-69.114,174.715,22.090,153.689
C02593=1082.629,138.972,-69.134,174.716,22.092,153.689
C02594=1082.635,139.221,-69.154,174.719,22.094,153.689
C02595=1082.640,139.470,-69.175,174.721,22.096,153.689
C02596=1082.645,139.719,-69.195,174.723,22.098,153.689
C02597=1082.651,139.969,-69.215,174.725,22.100,153.689
C02598=1082.656,140.218,-69.235,174.727,22.102,153.689
C02599=1082.662,140.467,-69.255,174.729,22.104,153.689
C02600=1082.668,140.717,-69.276,174.731,22.106,153.690
C02601=1082.674,140.965,-69.296,174.733,22.108,153.690
C02602=1082.679,141.215,-69.317,174.736,22.110,153.690
C02603=1082.685,141.464,-69.337,174.737,22.112,153.690
C02604=1082.691,141.713,-69.357,174.740,22.114,153.690
C02605=1082.696,141.962,-69.378,174.742,22.116,153.690
C02606=1082.701,142.211,-69.398,174.743,22.118,153.690
C02607=1082.707,142.460,-69.418,174.746,22.120,153.690
C02608=1082.713,142.709,-69.439,174.748,22.122,153.690
C02609=1082.718,142.959,-69.460,174.750,22.124,153.690
C02610=1082.725,143.238,-69.482,174.752,22.126,153.691
C02611=1082.731,143.517,-69.505,174.754,22.128,153.691
C02612=1082.737,143.797,-69.529,174.756,22.131,153.691
C02613=1082.744,144.077,-69.552,174.760,22.133,153.691
C02614=1082.749,144.326,-69.572,174.761,22.135,153.691
C02615=1082.755,144.575,-69.592,174.764,22.137,153.691
C02616=1082.760,144.824,-69.613,174.766,22.139,153.691
C02617=1082.765,145.073,-69.633,174.767,22.141,153.691
C02618=1082.771,145.322,-69.655,174.770,22.143,153.691
C02619=1082.778,145.571,-69.675,174.772,22.145,153.691
C02620=1082.783,145.820,-69.695,174.773,22.146,153.691
C02621=1082.788,146.069,-69.716,174.776,22.149,153.692
C02622=1082.793,146.318,-69.737,174.778,22.151,153.692
C02623=1082.799,146.567,-69.756,174.780,22.153,153.692
C02624=1082.806,146.816,-69.778,174.782,22.154,153.692
C02625=1082.811,147.066,-69.799,174.784,22.157,153.692
C02626=1082.817,147.314,-69.819,174.787,22.158,153.692
C02627=1082.822,147.563,-69.839,174.788,22.160,153.692
C02628=1082.828,147.813,-69.860,174.791,22.162,153.692
C02629=1082.833,148.062,-69.881,174.793,22.164,153.692
C02630=1082.839,148.311,-69.902,174.795,22.166,153.692
C02631=1082.845,148.560,-69.922,174.797,22.168,153.692
C02632=1082.851,148.810,-69.943,174.799,22.170,153.693
C02633=1082.856,149.058,-69.964,174.801,22.172,153.693
C02634=1082.861,149.307,-69.985,174.804,22.174,153.693
C02635=1082.867,149.556,-70.005,174.805,22.176,153.693
C02636=1082.873,149.806,-70.027,174.808,22.178,153.693
C02637=1082.878,150.055,-70.047,174.810,22.180,153.693
C02638=1082.883,150.304,-70.068,174.812,22.182,153.693
C02639=1082.890,150.552,-70.089,174.814,22.184,153.693
C02640=1082.895,150.802,-70.110,174.816,22.186,153.693
C02641=1082.901,151.051,-70.130,174.819,22.188,153.693
C02642=1082.906,151.299,-70.151,174.820,22.189,153.693
C02643=1082.912,151.549,-70.172,174.822,22.192,153.694
C02644=1082.917,151.798,-70.193,174.825,22.194,153.694
C02645=1082.923,152.047,-70.214,174.827,22.196,153.694
C02646=1082.928,152.296,-70.235,174.829,22.197,153.694
C02647=1082.934,152.545,-70.256,174.831,22.200,153.694
C02648=1082.940,152.794,-70.277,174.833,22.201,153.694
C02649=1082.945,153.043,-70.298,174.836,22.204,153.694
C02650=1082.951,153.293,-70.319,174.837,22.205,153.694
C02651=1082.956,153.542,-70.340,174.840,22.207,153.694
C02652=1082.962,153.790,-70.361,174.842,22.209,153.694
C02653=1082.968,154.040,-70.382,174.844,22.212,153.694
C02654=1082.973,154.289,-70.403,174.847,22.213,153.694
C02655=1082.979,154.538,-70.424,174.848,22.215,153.695
C02656=1082.985,154.787,-70.445,174.851,22.217,153.695
C02657=1082.990,155.036,-70.466,174.853,22.219,153.695
C02658=1082.995,155.285,-70.487,174.855,22.221,153.695
C02659=1083.002,155.534,-70.509,174.857,22.223,153.695
C02660=1083.007,155.783,-70.529,174.859,22.225,153.695
C02661=1083.012,156.031,-70.551,174.862,22.227,153.695
C02662=1083.018,156.281,-70.571,174.864,22.229,153.695
C02663=1083.024,156.530,-70.593,174.866,22.231,153.695
C02664=1083.029,156.779,-70.613,174.868,22.233,153.695
C02665=1083.035,157.028,-70.635,174.870,22.235,153.695
C02666=1083.041,157.277,-70.656,174.873,22.237,153.695
C02667=1083.045,157.526,-70.677,174.875,22.239,153.695
C02668=1083.052,157.775,-70.699,174.877,22.240,153.695
C02669=1083.057,158.024,-70.719,174.879,22.243,153.696
C02670=1083.063,158.274,-70.741,174.881,22.244,153.696
C02671=1083.069,158.522,-70.762,174.884,22.247,153.696
C02672=1083.074,158.771,-70.783,174.886,22.248,153.696
C02673=1083.080,159.020,-70.805,174.887,22.250,153.696
C02674=1083.086,159.299,-70.829,174.890,22.252,153.696
C02675=1083.092,159.580,-70.852,174.893,22.255,153.696
C02676=1083.098,159.859,-70.877,174.896,22.257,153.696
C02677=1083.105,160.137,-70.900,174.898,22.259,153.696
C02678=1083.110,160.387,-70.922,174.900,22.261,153.696
C02679=1083.116,160.636,-70.943,174.902,22.263,153.696
C02680=1083.122,160.885,-70.964,174.904,22.265,153.696
C02681=1083.127,161.134,-70.986,174.907,22.266,153.696
C02682=1083.133,161.383,-71.007,174.909,22.269,153.697
C02683=1083.139,161.631,-71.029,174.911,22.271,153.697
C02684=1083.144,161.881,-71.050,174.913,22.272,153.697
C02685=1083.150,162.130,-71.071,174.915,22.274,153.697
C02686=1083.155,162.379,-71.093,174.917,22.277,153.697
C02687=1083.160,162.627,-71.115,174.920,22.278,153.697
C02688=1083.166,162.877,-71.137,174.922,22.281,153.697
C02689=1083.171,163.126,-71.157,174.925,22.282,153.697
C02690=1083.177,163.375,-71.179,174.926,22.284,153.697
C02691=1083.182,163.624,-71.201,174.929,22.286,153.697
C02692=1083.187,163.873,-71.222,174.931,22.289,153.697
C02693=1083.193,164.122,-71.244,174.933,22.290,153.697
C02694=1083.198,164.371,-71.266,174.936,22.293,153.698
C02695=1083.204,164.620,-71.288,174.938,22.294,153.698
C02696=1083.209,164.869,-71.309,174.939,22.296,153.698
C02697=1083.214,165.118,-71.330,174.942,22.298,153.698
C02698=1083.220,165.367,-71.352,174.944,22.300,153.698
C02699=1083.225,165.616,-71.374,174.947,22.302,153.698
C02700=1083.231,165.865,-71.395,174.949,22.304,153.698
C02701=1083.236,166.114,-71.417,174.951,22.306,153.698
C02702=1083.242,166.363,-71.439,174.953,22.308,153.698
C02703=1083.247,166.612,-71.461,174.955,22.310,153.698
C02704=1083.253,166.861,-71.482,174.958,22.312,153.698
C02705=1083.258,167.110,-71.504,174.960,22.314,153.698
C02706=1083.264,167.359,-71.526,174.962,22.316,153.698
C02707=1083.269,167.608,-71.548,174.965,22.318,153.699
C02708=1083.275,167.857,-71.569,174.966,22.320,153.699
C02709=1083.280,168.106,-71.591,174.969,22.322,153.699
C02710=1083.286,168.355,-71.613,174.971,22.324,153.699
C02711=1083.291,168.604,-71.635,174.974,22.326,153.699
C02712=1083.297,168.853,-71.657,174.976,22.328,153.699
C02713=1083.302,169.102,-71.679,174.978,22.330,153.699
C02714=1083.308,169.351,-71.701,174.981,22.332,153.699
C02715=1083.313,169.600,-71.722,174.982,22.334,153.699
C02716=1083.319,169.849,-71.744,174.985,22.335,153.699
C02717=1083.324,170.098,-71.766,174.987,22.337,153.699
C02718=1083.330,170.347,-71.788,174.989,22.339,153.699
C02719=1083.335,170.596,-71.809,174.992,22.341,153.699
C02720=1083.341,170.844,-71.832,174.994,22.344,153.699
C02721=1083.347,171.094,-71.854,174.997,22.345,153.699
C02722=1083.352,171.343,-71.876,174.999,22.347,153.700
C02723=1083.358,171.592,-71.897,175.000,22.349,153.700
C02724=1083.363,171.841,-71.919,175.003,22.351,153.700
C02725=1083.369,172.089,-71.942,175.005,22.353,153.700
C02726=1083.375,172.339,-71.964,175.008,22.355,153.700
C02727=1083.380,172.587,-71.985,175.010,22.357,153.700
C02728=1083.386,172.837,-72.007,175.013,22.359,153.700
C02729=1083.390,173.086,-72.029,175.015,22.361,153.700
C02730=1083.397,173.334,-72.052,175.017,22.363,153.700
C02731=1083.402,173.584,-72.074,175.020,22.365,153.700
C02732=1083.408,173.832,-72.095,175.021,22.366,153.700
C02733=1083.414,174.081,-72.118,175.024,22.368,153.700
C02734=1083.419,174.331,-72.140,175.026,22.370,153.700
C02735=1083.425,174.579,-72.162,175.029,22.372,153.700
C02736=1083.430,174.828,-72.185,175.031,22.374,153.700
C02737=1083.436,175.078,-72.207,175.033,22.376,153.700
C02738=1083.442,175.357,-72.231,175.036,22.378,153.700
C02739=1083.448,175.635,-72.256,175.038,22.380,153.701
C02740=1083.455,175.914,-72.281,175.041,22.382,153.701
C02741=1083.461,176.193,-72.305,175.044,22.385,153.701
C02742=1083.467,176.442,-72.328,175.046,22.386,153.701
C02743=1083.472,176.691,-72.350,175.049,22.388,153.701
C02744=1083.478,176.940,-72.372,175.051,22.390,153.701
C02745=1083.483,177.189,-72.394,175.053,22.392,153.701
C02746=1083.489,177.438,-72.417,175.055,22.394,153.701
C02747=1083.495,177.687,-72.439,175.058,22.396,153.701
C02748=1083.500,177.936,-72.461,175.060,22.397,153.701
C02749=1083.506,178.185,-72.484,175.062,22.399,153.701
C02750=1083.512,178.434,-72.505,175.065,22.401,153.701
C02751=1083.518,178.683,-72.528,175.067,22.403,153.701
C02752=1083.522,178.932,-72.550,175.070,22.405,153.701
C02753=1083.529,179.180,-72.572,175.072,22.407,153.701
C02754=1083.534,179.430,-72.595,175.074,22.409,153.701
C02755=1083.540,179.679,-72.618,175.077,22.411,153.701
C02756=1083.546,179.928,-72.639,175.079,22.413,153.701
C02757=1083.551,180.176,-72.662,175.082,22.415,153.701
C02758=1083.557,180.425,-72.685,175.084,22.416,153.701
C02759=1083.563,180.674,-72.707,175.087,22.418,153.701
C02760=1083.569,180.923,-72.729,175.088,22.420,153.702
C02761=1083.574,181.172,-72.752,175.091,22.422,153.702
C02762=1083.580,181.421,-72.774,175.093,22.424,153.702
C02763=1083.586,181.669,-72.797,175.096,22.426,153.702
C02764=1083.591,181.919,-72.819,175.098,22.427,153.702
C02765=1083.597,182.168,-72.842,175.101,22.429,153.702
C02766=1083.603,182.417,-72.864,175.103,22.431,153.702
C02767=1083.609,182.666,-72.886,175.105,22.433,153.702
C02768=1083.614,182.914,-72.909,175.108,22.435,153.702
C02769=1083.620,183.163,-72.931,175.110,22.437,153.702
C02770=1083.625,183.412,-72.954,175.113,22.439,153.702
C02771=1083.632,183.661,-72.976,175.115,22.440,153.702
C02772=1083.638,183.910,-72.999,175.118,22.442,153.702
C02773=1083.643,184.159,-73.022,175.120,22.444,153.702
C02774=1083.649,184.408,-73.045,175.122,22.446,153.702
C02775=1083.654,184.657,-73.068,175.125,22.448,153.702
C02776=1083.660,184.905,-73.089,175.127,22.450,153.702
C02777=1083.666,185.155,-73.112,175.130,22.452,153.702
C02778=1083.671,185.403,-73.135,175.132,22.454,153.702
C02779=1083.677,185.652,-73.158,175.135,22.456,153.702
C02780=1083.682,185.902,-73.181,175.137,22.458,153.702
C02781=1083.687,186.150,-73.203,175.140,22.459,153.702
C02782=1083.693,186.399,-73.226,175.142,22.462,153.702
C02783=1083.698,186.648,-73.249,175.144,22.464,153.702
C02784=1083.704,186.897,-73.272,175.147,22.465,153.702
C02785=1083.710,187.146,-73.295,175.149,22.468,153.703
C02786=1083.715,187.394,-73.317,175.152,22.470,153.703
C02787=1083.720,187.643,-73.341,175.154,22.471,153.703
C02788=1083.725,187.893,-73.363,175.156,22.474,153.703
C02789=1083.731,188.142,-73.386,175.159,22.475,153.703
C02790=1083.737,188.391,-73.409,175.161,22.477,153.703
C02791=1083.742,188.639,-73.432,175.164,22.480,153.703
C02792=1083.748,188.888,-73.455,175.166,22.481,153.703
C02793=1083.753,189.137,-73.478,175.168,22.483,153.703
C02794=1083.759,189.386,-73.501,175.171,22.485,153.703
C02795=1083.764,189.635,-73.524,175.173,22.487,153.703
C02796=1083.770,189.884,-73.547,175.176,22.489,153.703
C02797=1083.776,190.133,-73.570,175.178,22.491,153.703
C02798=1083.780,190.381,-73.593,175.180,22.493,153.703
C02799=1083.786,190.630,-73.616,175.183,22.495,153.703
C02800=1083.792,190.879,-73.639,175.185,22.497,153.703
C02801=1083.797,191.128,-73.662,175.188,22.499,153.703
C02802=1083.803,191.407,-73.688,175.190,22.501,153.704
C02803=1083.809,191.685,-73.714,175.194,22.503,153.704
C02804=1083.817,191.964,-73.740,175.196,22.505,153.704
C02805=1083.822,192.242,-73.765,175.198,22.507,153.704
C02806=1083.827,192.492,-73.789,175.201,22.509,153.704
C02807=1083.833,192.741,-73.812,175.203,22.511,153.704
C02808=1083.839,192.989,-73.834,175.206,22.513,153.704
C02809=1083.845,193.238,-73.858,175.208,22.515,153.704
C02810=1083.850,193.487,-73.881,175.211,22.517,153.704
C02811=1083.855,193.736,-73.905,175.214,22.519,153.704
C02812=1083.861,193.985,-73.928,175.216,22.521,153.704
C02813=1083.867,194.234,-73.951,175.219,22.523,153.704
C02814=1083.872,194.483,-73.974,175.221,22.525,153.704
C02815=1083.877,194.732,-73.997,175.224,22.527,153.704
C02816=1083.884,194.980,-74.021,175.226,22.528,153.704
C02817=1083.889,195.229,-74.044,175.228,22.531,153.704
C02818=1083.894,195.478,-74.067,175.231,22.533,153.704
C02819=1083.900,195.727,-74.090,175.233,22.534,153.704
C02820=1083.906,195.975,-74.114,175.236,22.536,153.704
C02821=1083.912,196.224,-74.137,175.238,22.538,153.704
C02822=1083.917,196.473,-74.160,175.241,22.540,153.705
C02823=1083.922,196.722,-74.183,175.243,22.542,153.705
C02824=1083.928,196.971,-74.207,175.246,22.544,153.705
C02825=1083.933,197.220,-74.230,175.248,22.546,153.705
C02826=1083.939,197.469,-74.253,175.250,22.547,153.705
C02827=1083.945,197.717,-74.277,175.253,22.549,153.705
C02828=1083.950,197.966,-74.301,175.256,22.552,153.705
C02829=1083.956,198.215,-74.324,175.259,22.554,153.705
C02830=1083.963,198.464,-74.348,175.261,22.556,153.705
C02831=1083.968,198.713,-74.371,175.264,22.557,153.705
C02832=1083.973,198.962,-74.394,175.266,22.559,153.705
C02833=1083.979,199.210,-74.418,175.269,22.561,153.705
C02834=1083.984,199.460,-74.441,175.271,22.563,153.705
C02835=1083.990,199.708,-74.465,175.273,22.565,153.705
C02836=1083.996,199.957,-74.488,175.276,22.567,153.705
C02837=1084.001,200.206,-74.511,175.278,22.569,153.705
C02838=1084.007,200.454,-74.535,175.281,22.570,153.705
C02839=1084.013,200.704,-74.558,175.283,22.572,153.705
C02840=1084.019,200.952,-74.583,175.287,22.574,153.705
C02841=1084.025,201.201,-74.606,175.289,22.576,153.705
C02842=1084.030,201.450,-74.630,175.291,22.579,153.705
C02843=1084.036,201.699,-74.653,175.294,22.580,153.705
C02844=1084.042,201.947,-74.676,175.296,22.582,153.705
C02845=1084.047,202.196,-74.700,175.299,22.584,153.705
C02846=1084.053,202.445,-74.724,175.301,22.586,153.705
C02847=1084.058,202.694,-74.748,175.304,22.588,153.705
C02848=1084.064,202.943,-74.771,175.306,22.589,153.705
C02849=1084.069,203.192,-74.795,175.309,22.592,153.705
C02850=1084.075,203.440,-74.818,175.312,22.594,153.705
C02851=1084.081,203.689,-74.843,175.314,22.596,153.705
C02852=1084.086,203.938,-74.866,175.317,22.597,153.705
C02853=1084.092,204.187,-74.890,175.319,22.600,153.706
C02854=1084.097,204.436,-74.914,175.322,22.602,153.706
C02855=1084.103,204.684,-74.937,175.324,22.603,153.706
C02856=1084.109,204.933,-74.962,175.327,22.605,153.706
C02857=1084.114,205.182,-74.985,175.330,22.608,153.706
C02858=1084.120,205.431,-75.009,175.332,22.610,153.706
C02859=1084.125,205.679,-75.033,175.335,22.611,153.706
C02860=1084.130,205.929,-75.057,175.337,22.613,153.706
C02861=1084.137,206.177,-75.081,175.340,22.615,153.706
C02862=1084.142,206.426,-75.105,175.342,22.617,153.706
C02863=1084.147,206.674,-75.129,175.344,22.619,153.706
C02864=1084.153,206.923,-75.152,175.348,22.621,153.706
C02865=1084.159,207.173,-75.177,175.350,22.623,153.706
C02866=1084.182,208.202,-75.276,175.436,22.669,153.703
C02867=1084.191,208.592,-75.314,175.441,22.673,153.704
C02868=1084.200,208.984,-75.353,175.444,22.678,153.704
C02869=1084.209,209.375,-75.391,175.448,22.682,153.704
C02870=1084.217,209.765,-75.430,175.452,22.687,153.705
C02871=1084.223,210.015,-75.454,175.455,22.689,153.705
C02872=1084.228,210.263,-75.479,175.457,22.692,153.705
C02873=1084.234,210.511,-75.504,175.460,22.695,153.706
C02874=1084.240,210.760,-75.528,175.462,22.698,153.706
C02875=1084.246,211.009,-75.552,175.464,22.701,153.706
C02876=1084.252,211.258,-75.576,175.467,22.704,153.706
C02877=1084.257,211.506,-75.601,175.469,22.707,153.707
C02878=1084.263,211.755,-75.626,175.471,22.710,153.707
C02879=1084.268,212.004,-75.651,175.474,22.713,153.707
C02880=1084.274,212.253,-75.676,175.477,22.715,153.707
C02881=1084.279,212.501,-75.700,175.480,22.719,153.708
C02882=1084.285,212.750,-75.725,175.482,22.721,153.708
C02883=1084.291,212.999,-75.750,175.484,22.724,153.708
C02884=1084.296,213.247,-75.774,175.487,22.727,153.709
C02885=1084.302,213.497,-75.799,175.489,22.730,153.709
C02886=1084.308,213.745,-75.824,175.491,22.733,153.709
C02887=1084.313,213.994,-75.849,175.494,22.736,153.709
C02888=1084.319,214.242,-75.873,175.496,22.739,153.710
C02889=1084.325,214.491,-75.898,175.499,22.742,153.710
C02890=1084.329,214.740,-75.923,175.501,22.745,153.710
C02891=1084.336,214.989,-75.948,175.504,22.747,153.710
C02892=1084.341,215.237,-75.973,175.507,22.751,153.711
C02893=1084.347,215.486,-75.998,175.509,22.753,153.711
C02894=1084.352,215.735,-76.022,175.512,22.757,153.711
C02895=1084.358,215.984,-76.048,175.514,22.759,153.711
C02896=1084.363,216.232,-76.072,175.516,22.762,153.712
C02897=1084.369,216.481,-76.098,175.519,22.765,153.712
C02898=1084.375,216.729,-76.122,175.521,22.768,153.712
C02899=1084.381,216.978,-76.147,175.524,22.771,153.712
C02900=1084.386,217.227,-76.172,175.526,22.774,153.713
C02901=1084.392,217.476,-76.197,175.529,22.777,153.713
C02902=1084.398,217.725,-76.222,175.532,22.780,153.713
C02903=1084.403,217.973,-76.247,175.534,22.783,153.714
C02904=1084.409,218.222,-76.272,175.537,22.786,153.714
C02905=1084.414,218.470,-76.297,175.539,22.789,153.714
C02906=1084.420,218.719,-76.323,175.541,22.791,153.714
C02907=1084.426,218.968,-76.347,175.544,22.794,153.715
C02908=1084.432,219.216,-76.372,175.546,22.797,153.715
C02909=1084.437,219.465,-76.398,175.549,22.800,153.715
C02910=1084.442,219.714,-76.422,175.551,22.803,153.715
C02911=1084.449,219.963,-76.448,175.554,22.806,153.716
C02912=1084.455,220.211,-76.473,175.557,22.809,153.716
C02913=1084.459,220.460,-76.498,175.559,22.812,153.716
C02914=1084.466,220.709,-76.523,175.562,22.814,153.716
C02915=1084.472,220.958,-76.549,175.564,22.817,153.717
C02916=1084.477,221.206,-76.574,175.567,22.820,153.717
C02917=1084.483,221.455,-76.599,175.569,22.823,153.717
C02918=1084.488,221.703,-76.624,175.571,22.826,153.717
C02919=1084.498,222.098,-76.664,175.576,22.831,153.718
C02920=1084.507,222.493,-76.705,175.579,22.835,153.718
C02921=1084.515,222.888,-76.744,175.584,22.840,153.719
C02922=1084.524,223.283,-76.785,175.588,22.844,153.719
C02923=1084.530,223.532,-76.811,175.591,22.848,153.719
C02924=1084.535,223.780,-76.836,175.593,22.850,153.720
C02925=1084.541,224.029,-76.862,175.596,22.854,153.720
C02926=1084.547,224.277,-76.887,175.598,22.856,153.720
C02927=1084.552,224.526,-76.913,175.601,22.860,153.720
C02928=1084.558,224.774,-76.938,175.603,22.862,153.721
C02929=1084.563,225.024,-76.963,175.605,22.865,153.721
C02930=1084.569,225.272,-76.988,175.608,22.868,153.721
C02931=1084.574,225.521,-77.014,175.610,22.871,153.722
C02932=1084.580,225.770,-77.039,175.614,22.874,153.722
C02933=1084.586,226.019,-77.065,175.616,22.877,153.722
C02934=1084.592,226.266,-77.090,175.619,22.880,153.722
C02935=1084.597,226.515,-77.116,175.621,22.883,153.723
C02936=1084.602,226.764,-77.142,175.624,22.886,153.723
C02937=1084.609,227.013,-77.167,175.626,22.889,153.723
C02938=1084.614,227.261,-77.193,175.629,22.892,153.723
C02939=1084.620,227.509,-77.219,175.631,22.895,153.724
C02940=1084.626,227.758,-77.245,175.633,22.897,153.724
C02941=1084.632,228.007,-77.270,175.636,22.900,153.724
C02942=1084.637,228.255,-77.296,175.639,22.903,153.724
C02943=1084.643,228.504,-77.321,175.642,22.906,153.725
C02944=1084.648,228.753,-77.347,175.644,22.909,153.725
C02945=1084.654,229.002,-77.373,175.647,22.912,153.725
C02946=1084.660,229.251,-77.398,175.649,22.915,153.725
C02947=1084.665,229.500,-77.424,175.652,22.918,153.726
C02948=1084.671,229.747,-77.450,175.654,22.920,153.726
C02949=1084.677,229.996,-77.476,175.657,22.924,153.726
C02950=1084.682,230.245,-77.502,175.659,22.926,153.726
C02951=1084.688,230.494,-77.527,175.662,22.930,153.727
C02952=1084.694,230.742,-77.554,175.665,22.932,153.727
C02953=1084.699,230.990,-77.579,175.668,22.936,153.727
C02954=1084.705,231.239,-77.605,175.670,22.938,153.728
C02955=1084.711,231.488,-77.631,175.673,22.942,153.728
C02956=1084.717,231.736,-77.657,175.675,22.944,153.728
C02957=1084.722,231.985,-77.683,175.678,22.948,153.728
C02958=1084.727,232.234,-77.709,175.680,22.950,153.729
C02959=1084.733,232.482,-77.734,175.683,22.954,153.729
C02960=1084.739,232.731,-77.761,175.685,22.956,153.729
C02961=1084.744,232.980,-77.787,175.688,22.959,153.729
C02962=1084.750,233.228,-77.813,175.691,22.962,153.730
C02963=1084.756,233.477,-77.839,175.694,22.965,153.730
C02964=1084.762,233.726,-77.865,175.696,22.968,153.730
C02965=1084.768,233.974,-77.891,175.699,22.971,153.730
C02966=1084.773,234.223,-77.917,175.701,22.974,153.731
C02967=1084.778,234.471,-77.943,175.704,22.977,153.731
C02968=1084.784,234.720,-77.970,175.706,22.980,153.731
C02969=1084.789,234.969,-77.995,175.709,22.983,153.732
C02970=1084.795,235.217,-78.022,175.711,22.986,153.732
C02971=1084.804,235.603,-78.062,175.716,22.991,153.732
C02972=1084.813,235.989,-78.103,175.719,22.995,153.733
C02973=1084.822,236.376,-78.144,175.724,23.000,153.733
C02974=1084.830,236.762,-78.185,175.728,23.004,153.734
C02975=1084.836,237.011,-78.211,175.731,23.007,153.734
C02976=1084.841,237.260,-78.238,175.733,23.010,153.734
C02977=1084.847,237.509,-78.264,175.736,23.013,153.734
C02978=1084.853,237.756,-78.290,175.738,23.016,153.735
C02979=1084.858,238.005,-78.316,175.741,23.019,153.735
C02980=1084.864,238.253,-78.342,175.743,23.022,153.735
C02981=1084.870,238.502,-78.369,175.746,23.025,153.735
C02982=1084.875,238.751,-78.395,175.748,23.028,153.736
C02983=1084.881,238.999,-78.421,175.751,23.031,153.736
C02984=1084.887,239.247,-78.448,175.754,23.034,153.736
C02985=1084.892,239.496,-78.474,175.757,23.037,153.737
C02986=1084.898,239.745,-78.501,175.760,23.040,153.737
C02987=1084.904,239.993,-78.527,175.762,23.043,153.737
C02988=1084.909,240.242,-78.553,175.765,23.046,153.737
C02989=1084.915,240.490,-78.580,175.767,23.048,153.738
C02990=1084.921,240.739,-78.607,175.770,23.052,153.738
C02991=1084.927,240.987,-78.633,175.772,23.054,153.738
C02992=1084.932,241.237,-78.660,175.775,23.058,153.738
C02993=1084.938,241.485,-78.687,175.778,23.061,153.739
C02994=1084.944,241.734,-78.713,175.781,23.064,153.739
C02995=1084.949,241.982,-78.740,175.784,23.067,153.739
C02996=1084.955,242.231,-78.767,175.786,23.070,153.740
C02997=1084.961,242.479,-78.793,175.789,23.073,153.740
C02998=1084.966,242.728,-78.819,175.791,23.075,153.740
C02999=1084.972,242.976,-78.846,175.794,23.079,153.740
C03000=1084.978,243.225,-78.873,175.796,23.081,153.741
C03001=1084.984,243.473,-78.899,175.799,23.085,153.741
C03002=1084.989,243.722,-78.926,175.802,23.088,153.741
C03003=1084.994,243.970,-78.953,175.804,23.091,153.741
C03004=1085.000,244.218,-78.980,175.807,23.094,153.742
C03005=1085.006,244.467,-79.006,175.810,23.097,153.742
C03006=1085.011,244.715,-79.034,175.813,23.100,153.742
C03007=1085.017,244.964,-79.060,175.816,23.103,153.743
C03008=1085.023,245.213,-79.087,175.818,23.106,153.743
C03009=1085.028,245.461,-79.115,175.821,23.109,153.743
C03010=1085.034,245.710,-79.141,175.823,23.112,153.743
C03011=1085.040,245.958,-79.168,175.826,23.115,153.744
C03012=1085.046,246.207,-79.195,175.828,23.118,153.744
C03013=1085.051,246.455,-79.222,175.831,23.121,153.744
C03014=1085.056,246.704,-79.248,175.834,23.124,153.745
C03015=1085.062,246.952,-79.275,175.836,23.127,153.745
C03016=1085.068,247.201,-79.303,175.839,23.130,153.745
C03017=1085.074,247.450,-79.329,175.842,23.133,153.745
C03018=1085.079,247.698,-79.356,175.845,23.136,153.746
C03019=1085.084,247.947,-79.383,175.848,23.139,153.746
C03020=1085.090,248.194,-79.411,175.850,23.142,153.746
C03021=1085.096,248.443,-79.438,175.853,23.145,153.747
C03022=1085.101,248.691,-79.464,175.855,23.148,153.747
C03023=1085.109,249.072,-79.507,175.860,23.153,153.747
C03024=1085.118,249.451,-79.548,175.863,23.157,153.748
C03025=1085.126,249.830,-79.589,175.868,23.162,153.748
C03026=1085.135,250.210,-79.631,175.872,23.167,153.749
C03027=1085.141,250.458,-79.658,175.874,23.170,153.749
C03028=1085.146,250.707,-79.685,175.877,23.173,153.749
C03029=1085.151,250.955,-79.712,175.879,23.176,153.750
C03030=1085.158,251.204,-79.740,175.883,23.179,153.750
C03031=1085.163,251.452,-79.767,175.886,23.182,153.750
C03032=1085.169,251.701,-79.794,175.888,23.185,153.750
C03033=1085.174,251.949,-79.822,175.891,23.188,153.751
C03034=1085.180,252.197,-79.848,175.893,23.191,153.751
C03035=1085.186,252.447,-79.876,175.896,23.194,153.751
C03036=1085.192,252.694,-79.903,175.899,23.198,153.752
C03037=1085.197,252.943,-79.930,175.901,23.201,153.752
C03038=1085.202,253.191,-79.958,175.904,23.204,153.752
C03039=1085.208,253.440,-79.985,175.907,23.207,153.752
C03040=1085.214,253.688,-80.013,175.909,23.210,153.753
C03041=1085.220,253.936,-80.040,175.912,23.213,153.753
C03042=1085.225,254.185,-80.067,175.915,23.216,153.753
C03043=1085.231,254.434,-80.095,175.918,23.219,153.754
C03044=1085.236,254.682,-80.122,175.921,23.222,153.754
C03045=1085.242,254.930,-80.150,175.924,23.225,153.754
C03046=1085.247,255.179,-80.177,175.926,23.228,153.754
C03047=1085.253,255.427,-80.205,175.929,23.231,153.755
C03048=1085.259,255.675,-80.233,175.931,23.234,153.755
C03049=1085.264,255.924,-80.260,175.934,23.237,153.755
C03050=1085.270,256.173,-80.288,175.937,23.241,153.756
C03051=1085.276,256.421,-80.315,175.939,23.244,153.756
C03052=1085.282,256.669,-80.343,175.942,23.247,153.756
C03053=1085.287,256.918,-80.371,175.945,23.250,153.756
C03054=1085.293,257.166,-80.398,175.947,23.253,153.757
C03055=1085.299,257.415,-80.426,175.950,23.256,153.757
C03056=1085.304,257.664,-80.453,175.954,23.259,153.757
C03057=1085.310,257.911,-80.481,175.956,23.262,153.758
C03058=1085.316,258.160,-80.509,175.959,23.265,153.758
C03059=1085.322,258.408,-80.537,175.962,23.268,153.758
C03060=1085.327,258.656,-80.564,175.964,23.271,153.758
C03061=1085.333,258.905,-80.592,175.967,23.274,153.759
C03062=1085.339,259.153,-80.620,175.970,23.277,153.759
C03063=1085.345,259.402,-80.648,175.972,23.280,153.759
C03064=1085.350,259.650,-80.675,175.975,23.283,153.760
C03065=1085.356,259.899,-80.703,175.978,23.286,153.760
C03066=1085.362,260.147,-80.730,175.981,23.289,153.760
C03067=1085.368,260.395,-80.758,175.984,23.292,153.760
C03068=1085.374,260.644,-80.787,175.987,23.295,153.761
C03069=1085.379,260.892,-80.813,175.990,23.299,153.761
C03070=1085.385,261.141,-80.842,175.992,23.302,153.761
C03071=1085.391,261.389,-80.870,175.995,23.305,153.762
C03072=1085.397,261.638,-80.898,175.998,23.308,153.762
C03073=1085.403,261.885,-80.925,176.000,23.311,153.762
C03074=1085.409,262.134,-80.954,176.003,23.314,153.762
C03075=1085.417,262.511,-80.996,176.008,23.318,153.763
C03076=1085.426,262.888,-81.038,176.011,23.323,153.763
C03077=1085.435,263.264,-81.081,176.016,23.328,153.764
C03078=1085.443,263.640,-81.123,176.020,23.332,153.764
C03079=1085.450,263.889,-81.151,176.023,23.335,153.764
C03080=1085.456,264.137,-81.180,176.026,23.338,153.765
C03081=1085.461,264.385,-81.208,176.029,23.342,153.765
C03082=1085.467,264.634,-81.236,176.031,23.345,153.765
C03083=1085.473,264.882,-81.264,176.034,23.348,153.766
C03084=1085.478,265.131,-81.292,176.037,23.351,153.766
C03085=1085.484,265.379,-81.320,176.039,23.354,153.766
C03086=1085.490,265.628,-81.348,176.042,23.357,153.767
C03087=1085.495,265.876,-81.376,176.045,23.361,153.767
C03088=1085.501,266.125,-81.405,176.048,23.364,153.767
C03089=1085.507,266.372,-81.433,176.050,23.367,153.767
C03090=1085.513,266.621,-81.462,176.053,23.370,153.768
C03091=1085.518,266.869,-81.490,176.056,23.373,153.768
C03092=1085.524,267.118,-81.518,176.058,23.376,153.768
C03093=1085.529,267.366,-81.546,176.062,23.379,153.769
C03094=1085.534,267.615,-81.575,176.065,23.382,153.769
C03095=1085.540,267.862,-81.604,176.068,23.386,153.769
C03096=1085.546,268.111,-81.632,176.070,23.388,153.770
C03097=1085.552,268.360,-81.660,176.073,23.392,153.770
C03098=1085.557,268.608,-81.688,176.076,23.395,153.770
C03099=1085.564,268.856,-81.717,176.079,23.398,153.771
C03100=1085.569,269.104,-81.745,176.081,23.401,153.771
C03101=1085.575,269.353,-81.773,176.084,23.404,153.771
C03102=1085.581,269.601,-81.802,176.087,23.408,153.772
C03103=1085.586,269.849,-81.830,176.090,23.411,153.772
C03104=1085.592,270.098,-81.859,176.092,23.414,153.772
C03105=1085.597,270.345,-81.888,176.095,23.417,153.772
C03106=1085.603,270.594,-81.916,176.098,23.421,153.773
C03107=1085.610,270.842,-81.945,176.101,23.424,153.773
C03108=1085.615,271.090,-81.973,176.104,23.426,153.773
C03109=1085.620,271.339,-82.002,176.107,23.430,153.774
C03110=1085.626,271.587,-82.031,176.109,23.433,153.774
C03111=1085.632,271.835,-82.059,176.113,23.436,153.774
C03112=1085.638,272.084,-82.088,176.115,23.439,153.775
C03113=1085.643,272.332,-82.116,176.118,23.443,153.775
C03114=1085.649,272.580,-82.146,176.121,23.446,153.775
C03115=1085.655,272.829,-82.174,176.124,23.449,153.776
C03116=1085.660,273.076,-82.203,176.126,23.452,153.776
C03117=1085.666,273.325,-82.231,176.129,23.455,153.776
C03118=1085.672,273.573,-82.261,176.132,23.459,153.777
C03119=1085.677,273.822,-82.289,176.135,23.462,153.777
C03120=1085.683,274.070,-82.318,176.137,23.465,153.777
C03121=1085.689,274.318,-82.348,176.140,23.468,153.778
C03122=1085.694,274.566,-82.375,176.143,23.471,153.778
C03123=1085.700,274.814,-82.405,176.146,23.475,153.778
C03124=1085.706,275.063,-82.434,176.149,23.478,153.778
C03125=1085.711,275.311,-82.462,176.151,23.481,153.779
C03126=1085.717,275.559,-82.492,176.154,23.484,153.779
C03127=1085.726,275.939,-82.536,176.159,23.489,153.780
C03128=1085.734,276.318,-82.580,176.163,23.494,153.780
C03129=1085.743,276.698,-82.624,176.168,23.499,153.781
C03130=1085.752,277.078,-82.669,176.172,23.504,153.781
C03131=1085.758,277.325,-82.698,176.174,23.508,153.782
C03132=1085.764,277.574,-82.726,176.178,23.511,153.782
C03133=1085.769,277.822,-82.756,176.181,23.514,153.782
C03134=1085.775,278.070,-82.785,176.183,23.517,153.783
C03135=1085.780,278.318,-82.814,176.186,23.520,153.783
C03136=1085.787,278.566,-82.843,176.189,23.524,153.783
C03137=1085.792,278.815,-82.872,176.192,23.527,153.784
C03138=1085.798,279.064,-82.901,176.195,23.530,153.784
C03139=1085.804,279.312,-82.931,176.198,23.534,153.784
C03140=1085.809,279.559,-82.960,176.200,23.536,153.784
C03141=1085.815,279.808,-82.989,176.203,23.540,153.785
C03142=1085.821,280.056,-83.018,176.206,23.543,153.785
C03143=1085.826,280.304,-83.048,176.209,23.546,153.785
C03144=1085.833,280.553,-83.077,176.212,23.550,153.786
C03145=1085.838,280.800,-83.106,176.214,23.553,153.786
C03146=1085.843,281.049,-83.136,176.217,23.556,153.787
C03147=1085.849,281.297,-83.165,176.220,23.559,153.787
C03148=1085.855,281.545,-83.194,176.223,23.563,153.787
C03149=1085.861,281.793,-83.223,176.226,23.566,153.788
C03150=1085.867,282.042,-83.253,176.229,23.570,153.788
C03151=1085.872,282.290,-83.282,176.231,23.573,153.788
C03152=1085.877,282.538,-83.312,176.234,23.576,153.789
C03153=1085.883,282.786,-83.341,176.237,23.579,153.789
C03154=1085.889,283.035,-83.371,176.240,23.583,153.789
C03155=1085.894,283.283,-83.400,176.243,23.586,153.790
C03156=1085.901,283.531,-83.430,176.246,23.590,153.790
C03157=1085.906,283.778,-83.459,176.249,23.593,153.790
C03158=1085.911,284.027,-83.489,176.251,23.596,153.791
C03159=1085.917,284.275,-83.519,176.254,23.599,153.791
C03160=1085.923,284.523,-83.548,176.257,23.603,153.791
C03161=1085.929,284.772,-83.577,176.260,23.606,153.792
C03162=1085.934,285.020,-83.608,176.263,23.610,153.792
C03163=1085.941,285.268,-83.637,176.266,23.613,153.792
C03164=1085.946,285.516,-83.666,176.268,23.616,153.793
C03165=1085.952,285.765,-83.696,176.271,23.620,153.793
C03166=1085.957,286.012,-83.726,176.274,23.623,153.794
C03167=1085.962,286.260,-83.756,176.277,23.626,153.794
C03168=1085.969,286.508,-83.785,176.280,23.629,153.794
C03169=1085.975,286.756,-83.815,176.283,23.633,153.795
C03170=1085.980,287.005,-83.845,176.286,23.636,153.795
C03171=1085.986,287.253,-83.874,176.289,23.640,153.795
C03172=1085.992,287.501,-83.904,176.291,23.643,153.796
C03173=1085.998,287.749,-83.934,176.294,23.646,153.796
C03174=1086.003,287.997,-83.963,176.298,23.649,153.796
C03175=1086.009,288.245,-83.994,176.300,23.653,153.797
C03176=1086.014,288.494,-84.023,176.303,23.657,153.797
C03177=1086.020,288.741,-84.054,176.306,23.660,153.797
C03178=1086.026,288.990,-84.083,176.309,23.663,153.798
C03179=1086.036,289.379,-84.130,176.314,23.668,153.798
C03180=1086.044,289.768,-84.177,176.318,23.674,153.799
C03181=1086.053,290.157,-84.224,176.323,23.679,153.800
C03182=1086.062,290.546,-84.271,176.327,23.684,153.800
C03183=1086.068,290.794,-84.301,176.330,23.688,153.800
C03184=1086.073,291.042,-84.331,176.333,23.691,153.801
C03185=1086.080,291.291,-84.361,176.336,23.695,153.801
C03186=1086.085,291.539,-84.391,176.339,23.698,153.802
C03187=1086.091,291.787,-84.421,176.342,23.702,153.802
C03188=1086.097,292.035,-84.452,176.344,23.705,153.802
C03189=1086.102,292.283,-84.481,176.347,23.708,153.803
C03190=1086.108,292.531,-84.512,176.350,23.712,153.803
C03191=1086.114,292.779,-84.542,176.353,23.715,153.804
C03192=1086.120,293.027,-84.572,176.356,23.718,153.804
C03193=1086.125,293.275,-84.602,176.359,23.722,153.804
C03194=1086.131,293.523,-84.632,176.362,23.726,153.805
C03195=1086.137,293.771,-84.662,176.365,23.729,153.805
C03196=1086.143,294.019,-84.692,176.368,23.732,153.805
C03197=1086.148,294.267,-84.723,176.371,23.736,153.806
C03198=1086.153,294.515,-84.754,176.374,23.739,153.806
C03199=1086.159,294.763,-84.784,176.377,23.743,153.807
C03200=1086.165,295.012,-84.814,176.380,23.746,153.807
C03201=1086.171,295.260,-84.844,176.382,23.749,153.807
C03202=1086.177,295.508,-84.875,176.385,23.753,153.808
C03203=1086.183,295.756,-84.905,176.388,23.757,153.808
C03204=1086.189,296.003,-84.936,176.391,23.760,153.808
C03205=1086.195,296.251,-84.966,176.394,23.763,153.809
C03206=1086.200,296.499,-84.997,176.397,23.767,153.809
C03207=1086.206,296.748,-85.028,176.400,23.771,153.810
C03208=1086.212,296.996,-85.057,176.403,23.774,153.810
C03209=1086.217,297.244,-85.088,176.406,23.778,153.810
C03210=1086.223,297.492,-85.118,176.409,23.781,153.811
C03211=1086.228,297.740,-85.149,176.412,23.784,153.811
C03212=1086.234,297.988,-85.179,176.415,23.788,153.812
C03213=1086.240,298.236,-85.210,176.418,23.792,153.812
C03214=1086.246,298.485,-85.241,176.421,23.795,153.812
C03215=1086.251,298.732,-85.271,176.424,23.799,153.813
C03216=1086.256,298.981,-85.302,176.427,23.802,153.813
C03217=1086.263,299.228,-85.333,176.429,23.806,153.814
C03218=1086.268,299.476,-85.364,176.432,23.810,153.814
C03219=1086.273,299.724,-85.394,176.435,23.813,153.814
C03220=1086.279,299.972,-85.425,176.438,23.817,153.815
C03221=1086.285,300.220,-85.456,176.441,23.820,153.815
C03222=1086.291,300.468,-85.487,176.444,23.824,153.816
C03223=1086.296,300.716,-85.517,176.447,23.828,153.816
C03224=1086.302,300.964,-85.548,176.450,23.831,153.817
C03225=1086.307,301.212,-85.579,176.452,23.834,153.817
C03226=1086.313,301.460,-85.610,176.455,23.838,153.817
C03227=1086.319,301.708,-85.641,176.458,23.842,153.818
C03228=1086.324,301.956,-85.671,176.461,23.846,153.818
C03229=1086.330,302.204,-85.703,176.464,23.849,153.819
C03230=1086.336,302.451,-85.733,176.467,23.853,153.819
C03231=1086.345,302.854,-85.784,176.472,23.859,153.820
C03232=1086.354,303.258,-85.834,176.476,23.865,153.821
C03233=1086.363,303.661,-85.884,176.481,23.871,153.821
C03234=1086.373,304.065,-85.935,176.487,23.877,153.822
C03235=1086.379,304.313,-85.966,176.490,23.880,153.822
C03236=1086.384,304.561,-85.997,176.493,23.884,153.823
C03237=1086.389,304.808,-86.029,176.495,23.888,153.823
C03238=1086.396,305.057,-86.060,176.498,23.892,153.824
C03239=1086.401,305.305,-86.090,176.501,23.895,153.824
C03240=1086.407,305.552,-86.122,176.504,23.899,153.824
C03241=1086.413,305.801,-86.153,176.507,23.902,153.825
C03242=1086.419,306.048,-86.184,176.510,23.906,153.825
C03243=1086.424,306.296,-86.215,176.513,23.909,153.826
C03244=1086.430,306.544,-86.247,176.516,23.913,153.826
C03245=1086.436,306.792,-86.277,176.519,23.917,153.827
C03246=1086.442,307.041,-86.309,176.522,23.921,153.827
C03247=1086.448,307.288,-86.340,176.525,23.924,153.828
C03248=1086.453,307.536,-86.371,176.528,23.928,153.828
C03249=1086.459,307.784,-86.403,176.531,23.932,153.828
C03250=1086.465,308.032,-86.434,176.534,23.935,153.829
C03251=1086.471,308.280,-86.466,176.537,23.939,153.829
C03252=1086.477,308.527,-86.497,176.540,23.943,153.830
C03253=1086.482,308.775,-86.528,176.542,23.946,153.830
C03254=1086.488,309.024,-86.560,176.545,23.950,153.831
C03255=1086.494,309.271,-86.591,176.548,23.953,153.831
C03256=1086.500,309.520,-86.622,176.551,23.957,153.831
C03257=1086.505,309.767,-86.654,176.554,23.961,153.832
C03258=1086.512,310.015,-86.685,176.557,23.965,153.832
C03259=1086.517,310.263,-86.716,176.560,23.968,153.833
C03260=1086.523,310.511,-86.748,176.564,23.972,153.833
C03261=1086.529,310.759,-86.779,176.567,23.976,153.834
C03262=1086.535,311.007,-86.811,176.570,23.980,153.834
C03263=1086.540,311.254,-86.843,176.573,23.984,153.835
C03264=1086.546,311.503,-86.874,176.576,23.987,153.835
C03265=1086.552,311.750,-86.905,176.579,23.991,153.835
C03266=1086.558,311.999,-86.937,176.582,23.994,153.836
C03267=1086.564,312.246,-86.969,176.584,23.998,153.836
C03268=1086.570,312.494,-87.000,176.587,24.002,153.837
C03269=1086.576,312.742,-87.032,176.590,24.005,153.837
C03270=1086.582,312.990,-87.064,176.593,24.009,153.838
C03271=1086.587,313.239,-87.095,176.596,24.013,153.838
C03272=1086.593,313.486,-87.126,176.599,24.017,153.839
C03273=1086.599,313.734,-87.159,176.602,24.020,153.839
C03274=1086.605,313.982,-87.191,176.606,24.025,153.840
C03275=1086.611,314.230,-87.222,176.609,24.028,153.840
C03276=1086.618,314.478,-87.254,176.612,24.032,153.840
C03277=1086.623,314.725,-87.285,176.615,24.035,153.841
C03278=1086.629,314.973,-87.317,176.617,24.040,153.841
C03279=1086.635,315.222,-87.349,176.620,24.043,153.842
C03280=1086.640,315.469,-87.381,176.623,24.047,153.842
C03281=1086.646,315.717,-87.413,176.626,24.051,153.843
C03282=1086.651,315.964,-87.446,176.629,24.055,153.843
C03283=1086.661,316.371,-87.498,176.634,24.062,153.844
C03284=1086.670,316.777,-87.551,176.639,24.068,153.845
C03285=1086.680,317.183,-87.603,176.643,24.074,153.846
C03286=1086.689,317.589,-87.656,176.648,24.081,153.847
C03287=1086.694,317.837,-87.687,176.651,24.084,153.847
C03288=1086.700,318.085,-87.719,176.654,24.088,153.848
C03289=1086.705,318.332,-87.752,176.658,24.093,153.848
C03290=1086.711,318.581,-87.784,176.661,24.096,153.849
C03291=1086.717,318.829,-87.816,176.664,24.101,153.849
C03292=1086.723,319.076,-87.848,176.667,24.105,153.850
C03293=1086.729,319.324,-87.881,176.669,24.109,153.850
C03294=1086.734,319.572,-87.913,176.672,24.112,153.851
C03295=1086.739,319.820,-87.945,176.675,24.116,153.851
C03296=1086.746,320.068,-87.978,176.678,24.120,153.852
C03297=1086.752,320.316,-88.010,176.682,24.124,153.852
C03298=1086.757,320.563,-88.042,176.685,24.128,153.853
C03299=1086.763,320.811,-88.075,176.688,24.132,153.853
C03300=1086.769,321.059,-88.107,176.690,24.136,153.854
C03301=1086.774,321.306,-88.139,176.693,24.140,153.854
C03302=1086.780,321.555,-88.172,176.696,24.144,153.855
C03303=1086.786,321.802,-88.205,176.700,24.148,153.855
C03304=1086.792,322.051,-88.237,176.703,24.152,153.856
C03305=1086.797,322.298,-88.268,176.706,24.157,153.856
C03306=1086.803,322.546,-88.302,176.708,24.161,153.857
C03307=1086.809,322.794,-88.334,176.711,24.164,153.857
C03308=1086.815,323.042,-88.366,176.714,24.168,153.858
C03309=1086.820,323.289,-88.399,176.717,24.172,153.859
C03310=1086.826,323.537,-88.431,176.721,24.177,153.859
C03311=1086.832,323.785,-88.464,176.724,24.181,153.860
C03312=1086.838,324.033,-88.496,176.726,24.185,153.860
C03313=1086.844,324.281,-88.530,176.729,24.188,153.861
C03314=1086.849,324.528,-88.561,176.732,24.192,153.861
C03315=1086.856,324.776,-88.594,176.736,24.197,153.862
C03316=1086.861,325.024,-88.627,176.739,24.201,153.862
C03317=1086.867,325.272,-88.659,176.742,24.205,153.863
C03318=1086.873,325.520,-88.693,176.744,24.209,153.863
C03319=1086.879,325.768,-88.725,176.747,24.213,153.864
C03320=1086.885,326.015,-88.758,176.751,24.217,153.864
C03321=1086.890,326.263,-88.790,176.754,24.221,153.865
C03322=1086.896,326.511,-88.823,176.757,24.225,153.865
C03323=1086.902,326.758,-88.856,176.760,24.229,153.866
C03324=1086.908,327.006,-88.889,176.763,24.233,153.866
C03325=1086.914,327.254,-88.921,176.766,24.237,153.867
C03326=1086.920,327.502,-88.955,176.769,24.241,153.868
C03327=1086.926,327.750,-88.987,176.772,24.246,153.868
C03328=1086.932,327.997,-89.020,176.775,24.250,153.869
C03329=1086.938,328.245,-89.053,176.778,24.254,153.869
C03330=1086.944,328.493,-89.086,176.781,24.258,153.870
C03331=1086.949,328.741,-89.119,176.784,24.262,153.870
C03332=1086.956,328.989,-89.152,176.787,24.266,153.871
C03333=1086.961,329.237,-89.185,176.790,24.270,153.871
C03334=1086.967,329.485,-89.218,176.794,24.275,153.872
C03335=1086.977,329.883,-89.271,176.798,24.281,153.873
C03336=1086.987,330.283,-89.324,176.803,24.287,153.874
C03337=1086.996,330.682,-89.378,176.808,24.295,153.875
C03338=1087.006,331.081,-89.430,176.813,24.301,153.876
C03339=1087.012,331.330,-89.464,176.816,24.305,153.876
C03340=1087.018,331.577,-89.496,176.819,24.309,153.877
C03341=1087.024,331.825,-89.530,176.822,24.314,153.877
C03342=1087.029,332.073,-89.563,176.825,24.318,153.878
C03343=1087.036,332.320,-89.597,176.828,24.322,153.879
C03344=1087.041,332.568,-89.630,176.832,24.327,153.879
C03345=1087.047,332.816,-89.663,176.834,24.331,153.880
C03346=1087.053,333.064,-89.697,176.837,24.335,153.880
C03347=1087.059,333.311,-89.729,176.840,24.339,153.881
C03348=1087.064,333.559,-89.763,176.844,24.344,153.881
C03349=1087.070,333.806,-89.797,176.847,24.348,153.882
C03350=1087.076,334.054,-89.830,176.849,24.353,153.883
C03351=1087.081,334.302,-89.863,176.852,24.357,153.883
C03352=1087.088,334.550,-89.896,176.856,24.361,153.884
C03353=1087.094,334.797,-89.930,176.859,24.366,153.885
C03354=1087.099,335.045,-89.963,176.861,24.370,153.885
C03355=1087.105,335.293,-89.997,176.865,24.375,153.886
C03356=1087.110,335.540,-90.031,176.868,24.379,153.886
C03357=1087.117,335.788,-90.064,176.871,24.383,153.887
C03358=1087.122,336.036,-90.097,176.874,24.387,153.888
C03359=1087.129,336.284,-90.131,176.877,24.392,153.888
C03360=1087.134,336.532,-90.165,176.880,24.396,153.889
C03361=1087.140,336.779,-90.199,176.883,24.401,153.889
C03362=1087.147,337.026,-90.232,176.886,24.405,153.890
C03363=1087.152,337.274,-90.265,176.889,24.409,153.891
C03364=1087.158,337.522,-90.299,176.893,24.414,153.891
C03365=1087.163,337.770,-90.332,176.896,24.418,153.892
C03366=1087.170,338.018,-90.367,176.898,24.423,153.893
C03367=1087.175,338.265,-90.400,176.902,24.427,153.893
C03368=1087.181,338.513,-90.434,176.905,24.432,153.894
C03369=1087.187,338.760,-90.468,176.907,24.436,153.894
C03370=1087.193,339.008,-90.501,176.911,24.441,153.895
C03371=1087.199,339.255,-90.535,176.914,24.445,153.896
C03372=1087.204,339.503,-90.569,176.917,24.450,153.896
C03373=1087.211,339.751,-90.603,176.920,24.454,153.897
C03374=1087.217,339.998,-90.637,176.923,24.458,153.898
C03375=1087.222,340.246,-90.671,176.926,24.463,153.898
C03376=1087.228,340.494,-90.705,176.929,24.468,153.899
C03377=1087.234,340.741,-90.739,176.932,24.472,153.900
C03378=1087.240,340.989,-90.772,176.935,24.477,153.900
C03379=1087.246,341.237,-90.806,176.938,24.482,153.901
C03380=1087.252,341.484,-90.841,176.941,24.486,153.902
C03381=1087.258,341.731,-90.875,176.945,24.491,153.902
C03382=1087.262,341.979,-90.909,176.948,24.495,153.903
C03383=1087.269,342.227,-90.943,176.950,24.499,153.904
C03384=1087.275,342.475,-90.977,176.954,24.504,153.904
C03385=1087.281,342.722,-91.011,176.957,24.509,153.905
C03386=1087.287,342.970,-91.045,176.959,24.513,153.906
C03387=1087.295,343.364,-91.099,176.964,24.520,153.907
C03388=1087.306,343.757,-91.153,176.969,24.528,153.908
C03389=1087.314,344.150,-91.208,176.974,24.535,153.909
C03390=1087.324,344.544,-91.262,176.979,24.543,153.910
C03391=1087.330,344.792,-91.297,176.983,24.548,153.911
C03392=1087.336,345.039,-91.331,176.986,24.552,153.911
C03393=1087.342,345.287,-91.365,176.989,24.557,153.912
C03394=1087.348,345.534,-91.399,176.992,24.561,153.913
C03395=1087.354,345.782,-91.434,176.995,24.567,153.913
C03396=1087.359,346.029,-91.468,176.998,24.571,153.914
C03397=1087.365,346.277,-91.502,177.001,24.576,153.915
C03398=1087.371,346.525,-91.537,177.004,24.581,153.916
C03399=1087.377,346.772,-91.571,177.007,24.585,153.916
C03400=1087.383,347.020,-91.605,177.011,24.590,153.917
C03401=1087.388,347.268,-91.641,177.013,24.595,153.918
C03402=1087.395,347.515,-91.675,177.017,24.600,153.918
C03403=1087.400,347.762,-91.709,177.020,24.605,153.919
C03404=1087.406,348.010,-91.744,177.023,24.609,153.920
C03405=1087.412,348.257,-91.778,177.026,24.614,153.921
C03406=1087.418,348.505,-91.813,177.029,24.619,153.921
C03407=1087.424,348.752,-91.848,177.032,24.624,153.922
C03408=1087.430,349.000,-91.882,177.035,24.628,153.923
C03409=1087.436,349.248,-91.917,177.038,24.634,153.924
C03410=1087.442,349.495,-91.952,177.041,24.638,153.924
C03411=1087.447,349.743,-91.987,177.045,24.643,153.925
C03412=1087.453,349.990,-92.021,177.047,24.648,153.926
C03413=1087.460,350.238,-92.056,177.051,24.653,153.927
C03414=1087.465,350.485,-92.091,177.054,24.658,153.927
C03415=1087.471,350.732,-92.125,177.057,24.663,153.928
C03416=1087.477,350.980,-92.161,177.060,24.667,153.929
C03417=1087.483,351.227,-92.195,177.063,24.673,153.930
C03418=1087.489,351.475,-92.230,177.066,24.677,153.930
C03419=1087.495,351.722,-92.264,177.070,24.682,153.931
C03420=1087.501,351.970,-92.300,177.072,24.687,153.932
C03421=1087.507,352.217,-92.334,177.076,24.692,153.932
C03422=1087.513,352.465,-92.370,177.079,24.697,153.933
C03423=1087.519,352.712,-92.404,177.082,24.702,153.934
C03424=1087.525,352.960,-92.440,177.085,24.707,153.935
C03425=1087.530,353.207,-92.474,177.088,24.712,153.936
C03426=1087.536,353.455,-92.510,177.091,24.717,153.936
C03427=1087.542,353.703,-92.544,177.094,24.723,153.937
C03428=1087.548,353.950,-92.579,177.097,24.727,153.938
C03429=1087.554,354.197,-92.615,177.101,24.732,153.939
C03430=1087.560,354.445,-92.650,177.103,24.737,153.940
C03431=1087.566,354.693,-92.685,177.107,24.743,153.940
C03432=1087.572,354.940,-92.720,177.109,24.747,153.941
C03433=1087.577,355.188,-92.755,177.113,24.753,153.942
C03434=1087.584,355.434,-92.790,177.117,24.758,153.943
C03435=1087.590,355.682,-92.826,177.119,24.763,153.944
C03436=1087.595,355.929,-92.861,177.123,24.768,153.944
C03437=1087.601,356.177,-92.896,177.125,24.773,153.945
C03438=1087.607,356.424,-92.931,177.129,24.779,153.946
C03439=1087.617,356.821,-92.988,177.134,24.787,153.947
C03440=1087.626,357.216,-93.045,177.138,24.795,153.949
C03441=1087.635,357.614,-93.101,177.144,24.803,153.950
C03442=1087.645,358.009,-93.157,177.149,24.811,153.951
C03443=1087.651,358.257,-93.193,177.152,24.817,153.952
C03444=1087.657,358.505,-93.229,177.155,24.822,153.953
C03445=1087.663,358.752,-93.264,177.158,24.827,153.954
C03446=1087.669,358.999,-93.300,177.161,24.832,153.954
C03447=1087.675,359.247,-93.335,177.164,24.838,153.955
C03448=1087.681,359.494,-93.370,177.168,24.843,153.956
C03449=1087.687,359.741,-93.406,177.170,24.848,153.957
C03450=1087.693,359.989,-93.442,177.174,24.853,153.958
C03451=1087.699,360.237,-93.477,177.177,24.859,153.959
C03452=1087.704,360.484,-93.513,177.180,24.864,153.960
C03453=1087.711,360.731,-93.549,177.183,24.870,153.961
C03454=1087.717,360.978,-93.585,177.186,24.874,153.961
C03455=1087.723,361.225,-93.620,177.190,24.880,153.962
C03456=1087.729,361.473,-93.655,177.192,24.885,153.963
C03457=1087.735,361.720,-93.691,177.196,24.890,153.964
C03458=1087.740,361.967,-93.727,177.199,24.896,153.965
C03459=1087.747,362.214,-93.763,177.202,24.901,153.966
C03460=1087.753,362.462,-93.799,177.205,24.907,153.967
C03461=1087.759,362.710,-93.834,177.209,24.912,153.967
C03462=1087.764,362.957,-93.870,177.211,24.918,153.968
C03463=1087.770,363.204,-93.906,177.215,24.923,153.969
C03464=1087.776,363.451,-93.942,177.217,24.928,153.970
C03465=1087.783,363.699,-93.978,177.221,24.934,153.971
C03466=1087.789,363.946,-94.014,177.224,24.940,153.972
C03467=1087.794,364.193,-94.050,177.227,24.945,153.973
C03468=1087.801,364.440,-94.086,177.230,24.950,153.974
C03469=1087.807,364.688,-94.122,177.233,24.956,153.975
C03470=1087.812,364.936,-94.158,177.236,24.961,153.976
C03471=1087.818,365.183,-94.195,177.240,24.967,153.976
C03472=1087.824,365.430,-94.230,177.243,24.973,153.977
C03473=1087.830,365.677,-94.266,177.245,24.978,153.978
C03474=1087.836,365.925,-94.302,177.249,24.984,153.979
C03475=1087.842,366.172,-94.338,177.252,24.989,153.980
C03476=1087.848,366.420,-94.375,177.255,24.995,153.981
C03477=1087.853,366.666,-94.411,177.258,25.001,153.982
C03478=1087.860,366.913,-94.447,177.262,25.006,153.983
C03479=1087.866,367.161,-94.483,177.265,25.012,153.984
C03480=1087.871,367.408,-94.520,177.268,25.017,153.985
C03481=1087.878,367.655,-94.557,177.271,25.023,153.986
C03482=1087.884,367.903,-94.592,177.274,25.029,153.987
C03483=1087.889,368.149,-94.628,177.277,25.035,153.988
C03484=1087.895,368.396,-94.665,177.280,25.040,153.989
C03485=1087.901,368.644,-94.701,177.284,25.046,153.990
C03486=1087.907,368.891,-94.738,177.287,25.052,153.991
C03487=1087.913,369.139,-94.775,177.289,25.058,153.992
C03488=1087.919,369.386,-94.811,177.293,25.063,153.993
C03489=1087.925,369.633,-94.847,177.296,25.069,153.994
C03490=1087.932,369.880,-94.883,177.299,25.075,153.995
C03491=1087.941,370.292,-94.944,177.304,25.084,153.996
C03492=1087.952,370.704,-95.006,177.310,25.094,153.998
C03493=1087.961,371.116,-95.066,177.315,25.104,154.000
C03494=1087.972,371.528,-95.127,177.320,25.114,154.001
C03495=1087.978,371.775,-95.164,177.324,25.120,154.002
C03496=1087.983,372.022,-95.201,177.327,25.125,154.003
C03497=1087.990,372.269,-95.237,177.329,25.131,154.004
C03498=1087.996,372.516,-95.274,177.333,25.137,154.005
C03499=1088.002,372.764,-95.311,177.336,25.143,154.006
C03500=1088.008,373.011,-95.347,177.339,25.149,154.007
C03501=1088.014,373.258,-95.384,177.342,25.155,154.008
C03502=1088.020,373.505,-95.421,177.345,25.161,154.009
C03503=1088.026,373.752,-95.457,177.349,25.167,154.010
C03504=1088.032,374.000,-95.494,177.352,25.173,154.011
C03505=1088.039,374.246,-95.531,177.355,25.179,154.012
C03506=1088.044,374.493,-95.568,177.358,25.185,154.014
C03507=1088.050,374.741,-95.605,177.361,25.191,154.015
C03508=1088.056,374.988,-95.642,177.364,25.197,154.016
C03509=1088.062,375.235,-95.679,177.368,25.203,154.017
C03510=1088.068,375.482,-95.717,177.371,25.210,154.018
C03511=1088.074,375.729,-95.753,177.373,25.215,154.019
C03512=1088.080,375.976,-95.790,177.377,25.222,154.020
C03513=1088.085,376.223,-95.828,177.380,25.228,154.021
C03514=1088.092,376.470,-95.864,177.383,25.234,154.022
C03515=1088.097,376.718,-95.901,177.387,25.241,154.023
C03516=1088.104,376.964,-95.939,177.390,25.247,154.024
C03517=1088.110,377.212,-95.976,177.392,25.253,154.025
C03518=1088.116,377.459,-96.013,177.396,25.259,154.026
C03519=1088.122,377.706,-96.051,177.399,25.265,154.028
C03520=1088.128,377.953,-96.087,177.402,25.272,154.029
C03521=1088.134,378.200,-96.125,177.406,25.278,154.030
C03522=1088.140,378.447,-96.162,177.409,25.284,154.031
C03523=1088.146,378.694,-96.199,177.412,25.291,154.032
C03524=1088.152,378.941,-96.236,177.415,25.296,154.033
C03525=1088.158,379.189,-96.274,177.418,25.303,154.034
C03526=1088.164,379.436,-96.311,177.421,25.309,154.035
C03527=1088.171,379.682,-96.348,177.425,25.315,154.036
C03528=1088.176,379.929,-96.386,177.428,25.322,154.038
C03529=1088.182,380.177,-96.423,177.431,25.328,154.039
C03530=1088.189,380.424,-96.461,177.434,25.335,154.040
C03531=1088.195,380.670,-96.499,177.438,25.341,154.041
C03532=1088.201,380.918,-96.536,177.441,25.348,154.042
C03533=1088.207,381.164,-96.573,177.444,25.354,154.043
C03534=1088.213,381.412,-96.611,177.447,25.360,154.044
C03535=1088.220,381.658,-96.649,177.450,25.367,154.046
C03536=1088.225,381.906,-96.686,177.453,25.373,154.047
C03537=1088.231,382.152,-96.723,177.456,25.380,154.048
C03538=1088.238,382.400,-96.762,177.460,25.386,154.049
C03539=1088.244,382.647,-96.799,177.463,25.393,154.050
C03540=1088.250,382.893,-96.837,177.466,25.399,154.052
C03541=1088.255,383.141,-96.874,177.469,25.406,154.053
C03542=1088.262,383.388,-96.912,177.472,25.413,154.054
C03543=1088.268,383.608,-96.946,177.475,25.418,154.055
C03544=1088.273,383.828,-96.980,177.478,25.425,154.056
C03545=1088.278,384.047,-97.013,177.481,25.430,154.057
C03546=1088.283,384.267,-97.048,177.484,25.436,154.058
C03547=1088.289,384.487,-97.080,177.486,25.443,154.059
C03548=1088.294,384.707,-97.114,177.489,25.448,154.061
C03549=1088.300,384.927,-97.148,177.492,25.455,154.062
C03550=1088.305,385.146,-97.182,177.495,25.460,154.063
C03551=1088.311,385.393,-97.220,177.498,25.467,154.064
C03552=1088.317,385.641,-97.258,177.501,25.474,154.065
C03553=1088.323,385.887,-97.296,177.504,25.481,154.066
C03554=1088.329,386.135,-97.334,177.508,25.487,154.068
C03555=1088.335,386.382,-97.372,177.511,25.494,154.069
C03556=1088.342,386.628,-97.410,177.514,25.501,154.070
C03557=1088.348,386.875,-97.448,177.517,25.508,154.071
C03558=1088.353,387.122,-97.487,177.520,25.515,154.073
C03559=1088.359,387.369,-97.524,177.524,25.522,154.074
C03560=1088.366,387.616,-97.562,177.527,25.528,154.075
C03561=1088.372,387.862,-97.601,177.530,25.535,154.077
C03562=1088.378,388.110,-97.639,177.533,25.542,154.078
C03563=1088.384,388.357,-97.677,177.536,25.549,154.079
C03564=1088.390,388.603,-97.715,177.539,25.556,154.080
C03565=1088.396,388.851,-97.754,177.543,25.563,154.082
C03566=1088.402,389.097,-97.792,177.547,25.571,154.083
C03567=1088.409,389.344,-97.831,177.550,25.577,154.084
C03568=1088.415,389.591,-97.868,177.553,25.584,154.086
C03569=1088.422,389.838,-97.907,177.556,25.591,154.087
C03570=1088.428,390.084,-97.945,177.559,25.598,154.088
C03571=1088.433,390.332,-97.984,177.562,25.605,154.090
C03572=1088.440,390.578,-98.022,177.566,25.613,154.091
C03573=1088.446,390.826,-98.060,177.569,25.620,154.092
C03574=1088.452,391.072,-98.099,177.572,25.627,154.093
C03575=1088.459,391.319,-98.137,177.575,25.634,154.095
C03576=1088.464,391.566,-98.176,177.578,25.641,154.096
C03577=1088.471,391.813,-98.215,177.581,25.648,154.097
C03578=1088.478,392.060,-98.253,177.584,25.655,154.099
C03579=1088.483,392.306,-98.292,177.589,25.663,154.100
C03580=1088.490,392.553,-98.331,177.592,25.670,154.102
C03581=1088.496,392.800,-98.368,177.595,25.677,154.103
C03582=1088.502,393.047,-98.408,177.598,25.684,154.104
C03583=1088.508,393.293,-98.446,177.601,25.692,154.106
C03584=1088.514,393.541,-98.485,177.604,25.699,154.107
C03585=1088.521,393.788,-98.524,177.607,25.706,154.109
C03586=1088.526,394.034,-98.563,177.610,25.714,154.110
C03587=1088.533,394.281,-98.602,177.614,25.721,154.111
C03588=1088.539,394.529,-98.641,177.617,25.729,154.113
C03589=1088.545,394.775,-98.679,177.620,25.736,154.114
C03590=1088.551,395.022,-98.718,177.624,25.743,154.116
C03591=1088.558,395.269,-98.757,177.627,25.751,154.117
C03592=1088.563,395.515,-98.796,177.630,25.758,154.118
C03593=1088.570,395.762,-98.835,177.633,25.766,154.120
C03594=1088.576,396.009,-98.875,177.637,25.774,154.121
C03595=1088.582,396.256,-98.914,177.640,25.781,154.123
C03596=1088.588,396.503,-98.953,177.643,25.789,154.124
C03597=1088.595,396.750,-98.992,177.646,25.796,154.126
C03598=1088.601,396.996,-99.030,177.649,25.804,154.127
C03599=1088.606,397.223,-99.066,177.652,25.811,154.129
C03600=1088.612,397.450,-99.102,177.655,25.818,154.130
C03601=1088.617,397.676,-99.139,177.658,25.825,154.131
C03602=1088.624,397.903,-99.174,177.661,25.832,154.133
C03603=1088.629,398.130,-99.210,177.664,25.839,154.134
C03604=1088.635,398.356,-99.247,177.667,25.846,154.135
C03605=1088.640,398.583,-99.283,177.670,25.854,154.137
C03606=1088.647,398.810,-99.318,177.673,25.861,154.138
C03607=1088.653,399.057,-99.358,177.676,25.869,154.140
C03608=1088.658,399.302,-99.398,177.679,25.876,154.141
C03609=1088.665,399.550,-99.437,177.682,25.884,154.143
C03610=1088.671,399.796,-99.476,177.686,25.893,154.144
C03611=1088.677,400.044,-99.515,177.689,25.900,154.146
C03612=1088.684,400.290,-99.555,177.692,25.908,154.147
C03613=1088.689,400.537,-99.594,177.695,25.916,154.149
C03614=1088.695,400.784,-99.634,177.699,25.924,154.151
C03615=1088.702,401.030,-99.674,177.702,25.932,154.152
C03616=1088.709,401.277,-99.713,177.705,25.940,154.154
C03617=1088.715,401.524,-99.753,177.708,25.948,154.155
C03618=1088.721,401.771,-99.792,177.712,25.956,154.157
C03619=1088.727,402.018,-99.832,177.715,25.964,154.159
C03620=1088.733,402.264,-99.872,177.718,25.972,154.160
C03621=1088.740,402.511,-99.911,177.722,25.981,154.162
C03622=1088.746,402.758,-99.952,177.725,25.989,154.163
C03623=1088.752,403.005,-99.991,177.728,25.997,154.165
C03624=1088.758,403.251,-100.031,177.732,26.005,154.167
C03625=1088.764,403.497,-100.071,177.735,26.013,154.168
C03626=1088.771,403.744,-100.110,177.738,26.022,154.170
C03627=1088.777,403.991,-100.150,177.742,26.030,154.171
C03628=1088.783,404.238,-100.189,177.744,26.038,154.173
C03629=1088.790,404.484,-100.230,177.748,26.046,154.175
C03630=1088.796,404.731,-100.270,177.751,26.055,154.176
C03631=1088.803,404.977,-100.310,177.754,26.063,154.178
C03632=1088.808,405.225,-100.350,177.758,26.072,154.180
C03633=1088.814,405.471,-100.390,177.761,26.080,154.181
C03634=1088.821,405.719,-100.431,177.764,26.088,154.183
C03635=1088.828,405.965,-100.471,177.768,26.097,154.185
C03636=1088.834,406.212,-100.510,177.771,26.105,154.187
C03637=1088.840,406.459,-100.550,177.774,26.114,154.188
C03638=1088.846,406.705,-100.590,177.777,26.122,154.190
C03639=1088.853,406.952,-100.631,177.781,26.131,154.192
